    TriggL T1705,vl,laserOFF,z0,toolEtna\WObj:=wobjEtna;
    TriggL T1706,v50,laserON,z0,toolEtna\WObj:=wobjEtna;
    TriggL T1707,vl,laserOFF,z0,toolEtna\WObj:=wobjEtna;
    TriggL T1708,v50,laserON,z0,toolEtna\WObj:=wobjEtna;
    TriggL T1709,vl,laserOFF,z0,toolEtna\WObj:=wobjEtna;
    TriggL T1710,v50,laserON,z0,toolEtna\WObj:=wobjEtna;
    TriggL T1711,vl,laserOFF,z0,toolEtna\WObj:=wobjEtna;
    TriggL T1712,v50,laserON,z0,toolEtna\WObj:=wobjEtna;
    TriggL T1713,vl,laserOFF,z0,toolEtna\WObj:=wobjEtna;
    TriggL T1714,v50,laserON,z0,toolEtna\WObj:=wobjEtna;
    TriggL T1715,vl,laserOFF,z0,toolEtna\WObj:=wobjEtna;
    TriggL T1716,v50,laserON,z0,toolEtna\WObj:=wobjEtna;
    TriggL T1717,vl,laserOFF,z0,toolEtna\WObj:=wobjEtna;
    TriggL T1718,v50,laserON,z0,toolEtna\WObj:=wobjEtna;
    TriggL T1719,vl,laserOFF,z0,toolEtna\WObj:=wobjEtna;
    TriggL T1720,v50,laserON,z0,toolEtna\WObj:=wobjEtna;
    TriggL T1721,vl,laserOFF,z0,toolEtna\WObj:=wobjEtna;
    TriggL T1722,v50,laserON,z0,toolEtna\WObj:=wobjEtna;
    TriggL T1723,vl,laserOFF,z0,toolEtna\WObj:=wobjEtna;
    TriggL T1724,v50,laserON,z0,toolEtna\WObj:=wobjEtna;
    TriggL T1725,vl,laserOFF,z0,toolEtna\WObj:=wobjEtna;
    TriggL T1726,v50,laserON,z0,toolEtna\WObj:=wobjEtna;
    TriggL T1727,vl,laserOFF,z0,toolEtna\WObj:=wobjEtna;
    TriggL T1728,v50,laserON,z0,toolEtna\WObj:=wobjEtna;
    TriggL T1729,vl,laserOFF,z0,toolEtna\WObj:=wobjEtna;
    TriggL T1730,v50,laserON,z0,toolEtna\WObj:=wobjEtna;
    TriggL T1731,vl,laserOFF,z0,toolEtna\WObj:=wobjEtna;
    TriggL T1732,v50,laserON,z0,toolEtna\WObj:=wobjEtna;
    TriggL T1733,vl,laserOFF,z0,toolEtna\WObj:=wobjEtna;
    TriggL T1734,v50,laserON,z0,toolEtna\WObj:=wobjEtna;
    TriggL T1735,vl,laserOFF,z0,toolEtna\WObj:=wobjEtna;
    TriggL T1736,v50,laserON,z0,toolEtna\WObj:=wobjEtna;
    TriggL T1737,vl,laserOFF,z0,toolEtna\WObj:=wobjEtna;
    TriggL T1738,v50,laserON,z0,toolEtna\WObj:=wobjEtna;
    TriggL T1739,vl,laserOFF,z0,toolEtna\WObj:=wobjEtna;
    TriggL T1740,v50,laserON,z0,toolEtna\WObj:=wobjEtna;
    TriggL T1741,vl,laserOFF,z0,toolEtna\WObj:=wobjEtna;
    TriggL T1742,v50,laserON,z0,toolEtna\WObj:=wobjEtna;
    TriggL T1743,vl,laserOFF,z0,toolEtna\WObj:=wobjEtna;
    TriggL T1744,v50,laserON,z0,toolEtna\WObj:=wobjEtna;
    TriggL T1745,vl,laserOFF,z0,toolEtna\WObj:=wobjEtna;
    TriggL T1746,v50,laserON,z0,toolEtna\WObj:=wobjEtna;
    TriggL T1747,vl,laserOFF,z0,toolEtna\WObj:=wobjEtna;
    TriggL T1748,v50,laserON,z0,toolEtna\WObj:=wobjEtna;
    TriggL T1749,vl,laserOFF,z0,toolEtna\WObj:=wobjEtna;
    TriggL T1750,v50,laserON,z0,toolEtna\WObj:=wobjEtna;
    TriggL T1751,vl,laserOFF,z0,toolEtna\WObj:=wobjEtna;
    TriggL T1752,v50,laserON,z0,toolEtna\WObj:=wobjEtna;
    TriggL T1753,vl,laserOFF,z0,toolEtna\WObj:=wobjEtna;
    TriggL T1754,v50,laserON,z0,toolEtna\WObj:=wobjEtna;
    TriggL T1755,vl,laserOFF,z0,toolEtna\WObj:=wobjEtna;
    TriggL T1756,v50,laserON,z0,toolEtna\WObj:=wobjEtna;
    TriggL T1757,vl,laserOFF,z0,toolEtna\WObj:=wobjEtna;
    TriggL T1758,v50,laserON,z0,toolEtna\WObj:=wobjEtna;
    TriggL T1759,vl,laserOFF,z0,toolEtna\WObj:=wobjEtna;
    TriggL T1760,v50,laserON,z0,toolEtna\WObj:=wobjEtna;
    TriggL T1761,vl,laserOFF,z0,toolEtna\WObj:=wobjEtna;
    TriggL T1762,v50,laserON,z0,toolEtna\WObj:=wobjEtna;
    TriggL T1763,vl,laserOFF,z0,toolEtna\WObj:=wobjEtna;
    TriggL T1764,v50,laserON,z0,toolEtna\WObj:=wobjEtna;
    TriggL T1765,vl,laserOFF,z0,toolEtna\WObj:=wobjEtna;
    TriggL T1766,v50,laserON,z0,toolEtna\WObj:=wobjEtna;
    TriggL T1767,vl,laserOFF,z0,toolEtna\WObj:=wobjEtna;
    TriggL T1768,v50,laserON,z0,toolEtna\WObj:=wobjEtna;
    TriggL T1769,vl,laserOFF,z0,toolEtna\WObj:=wobjEtna;
    TriggL T1770,v50,laserON,z0,toolEtna\WObj:=wobjEtna;
    TriggL T1771,vl,laserOFF,z0,toolEtna\WObj:=wobjEtna;
    TriggL T1772,v50,laserON,z0,toolEtna\WObj:=wobjEtna;
    TriggL T1773,vl,laserOFF,z0,toolEtna\WObj:=wobjEtna;
    TriggL T1774,v50,laserON,z0,toolEtna\WObj:=wobjEtna;
    TriggL T1775,vl,laserOFF,z0,toolEtna\WObj:=wobjEtna;
    TriggL T1776,v50,laserON,z0,toolEtna\WObj:=wobjEtna;
    TriggL T1777,vl,laserOFF,z0,toolEtna\WObj:=wobjEtna;
    TriggL T1778,v50,laserON,z0,toolEtna\WObj:=wobjEtna;
    TriggL T1779,vl,laserOFF,z0,toolEtna\WObj:=wobjEtna;
    TriggL T1780,v50,laserON,z0,toolEtna\WObj:=wobjEtna;
    TriggL T1781,vl,laserOFF,z0,toolEtna\WObj:=wobjEtna;
    TriggL T1782,v50,laserON,z0,toolEtna\WObj:=wobjEtna;
    TriggL T1783,vl,laserOFF,z0,toolEtna\WObj:=wobjEtna;
    TriggL T1784,v50,laserON,z0,toolEtna\WObj:=wobjEtna;
    TriggL T1785,vl,laserOFF,z0,toolEtna\WObj:=wobjEtna;
    TriggL T1786,v50,laserON,z0,toolEtna\WObj:=wobjEtna;
    TriggL T1787,vl,laserOFF,z0,toolEtna\WObj:=wobjEtna;
    TriggL T1788,v50,laserON,z0,toolEtna\WObj:=wobjEtna;
    TriggL T1789,vl,laserOFF,z0,toolEtna\WObj:=wobjEtna;
    TriggL T1790,v50,laserON,z0,toolEtna\WObj:=wobjEtna;
    TriggL T1791,vl,laserOFF,z0,toolEtna\WObj:=wobjEtna;
    TriggL T1792,v50,laserON,z0,toolEtna\WObj:=wobjEtna;
    TriggL T1793,vl,laserOFF,z0,toolEtna\WObj:=wobjEtna;
    TriggL T1794,v50,laserON,z0,toolEtna\WObj:=wobjEtna;
    TriggL T1795,vl,laserOFF,z0,toolEtna\WObj:=wobjEtna;
    TriggL T1796,v50,laserON,z0,toolEtna\WObj:=wobjEtna;
    TriggL T1797,vl,laserOFF,z0,toolEtna\WObj:=wobjEtna;
    TriggL T1798,v50,laserON,z0,toolEtna\WObj:=wobjEtna;
    TriggL T1799,vl,laserOFF,z0,toolEtna\WObj:=wobjEtna;
    TriggL T1800,v50,laserON,z0,toolEtna\WObj:=wobjEtna;
    TriggL T1801,vl,laserOFF,z0,toolEtna\WObj:=wobjEtna;
    TriggL T1802,v50,laserON,z0,toolEtna\WObj:=wobjEtna;
    TriggL T1803,vl,laserOFF,z0,toolEtna\WObj:=wobjEtna;
    TriggL T1804,v50,laserON,z0,toolEtna\WObj:=wobjEtna;
    TriggL T1805,vl,laserOFF,z0,toolEtna\WObj:=wobjEtna;
    TriggL T1806,v50,laserON,z0,toolEtna\WObj:=wobjEtna;
    TriggL T1807,vl,laserOFF,z0,toolEtna\WObj:=wobjEtna;
    TriggL T1808,v50,laserON,z0,toolEtna\WObj:=wobjEtna;
    TriggL T1809,vl,laserOFF,z0,toolEtna\WObj:=wobjEtna;
    TriggL T1810,v50,laserON,z0,toolEtna\WObj:=wobjEtna;
    TriggL T1811,vl,laserOFF,z0,toolEtna\WObj:=wobjEtna;
    TriggL T1812,v50,laserON,z0,toolEtna\WObj:=wobjEtna;
    TriggL T1813,vl,laserOFF,z0,toolEtna\WObj:=wobjEtna;
    TriggL T1814,v50,laserON,z0,toolEtna\WObj:=wobjEtna;
    TriggL T1815,vl,laserOFF,z0,toolEtna\WObj:=wobjEtna;
    TriggL T1816,v50,laserON,z0,toolEtna\WObj:=wobjEtna;
    TriggL T1817,vl,laserOFF,z0,toolEtna\WObj:=wobjEtna;
    TriggL T1818,v50,laserON,z0,toolEtna\WObj:=wobjEtna;
    TriggL T1819,vl,laserOFF,z0,toolEtna\WObj:=wobjEtna;
    TriggL T1820,v50,laserON,z0,toolEtna\WObj:=wobjEtna;
    TriggL T1821,vl,laserOFF,z0,toolEtna\WObj:=wobjEtna;
    TriggL T1822,v50,laserON,z0,toolEtna\WObj:=wobjEtna;
    TriggL T1823,vl,laserOFF,z0,toolEtna\WObj:=wobjEtna;
    TriggL T1824,v50,laserON,z0,toolEtna\WObj:=wobjEtna;
    TriggL T1825,vl,laserOFF,z0,toolEtna\WObj:=wobjEtna;
    TriggL T1826,v50,laserON,z0,toolEtna\WObj:=wobjEtna;
    TriggL T1827,vl,laserOFF,z0,toolEtna\WObj:=wobjEtna;
    TriggL T1828,v50,laserON,z0,toolEtna\WObj:=wobjEtna;
    TriggL T1829,vl,laserOFF,z0,toolEtna\WObj:=wobjEtna;
    TriggL T1830,v50,laserON,z0,toolEtna\WObj:=wobjEtna;
    TriggL T1831,vl,laserOFF,z0,toolEtna\WObj:=wobjEtna;
    TriggL T1832,v50,laserON,z0,toolEtna\WObj:=wobjEtna;
    TriggL T1833,vl,laserOFF,z0,toolEtna\WObj:=wobjEtna;
    TriggL T1834,v50,laserON,z0,toolEtna\WObj:=wobjEtna;
    TriggL T1835,vl,laserOFF,z0,toolEtna\WObj:=wobjEtna;
    TriggL T1836,v50,laserON,z0,toolEtna\WObj:=wobjEtna;
    TriggL T1837,vl,laserOFF,z0,toolEtna\WObj:=wobjEtna;
    TriggL T1838,v50,laserON,z0,toolEtna\WObj:=wobjEtna;
    TriggL T1839,vl,laserOFF,z0,toolEtna\WObj:=wobjEtna;
    TriggL T1840,v50,laserON,z0,toolEtna\WObj:=wobjEtna;
    TriggL T1841,vl,laserOFF,z0,toolEtna\WObj:=wobjEtna;
    TriggL T1842,v50,laserON,z0,toolEtna\WObj:=wobjEtna;
    TriggL T1843,vl,laserOFF,z0,toolEtna\WObj:=wobjEtna;
    TriggL T1844,v50,laserON,z0,toolEtna\WObj:=wobjEtna;
    TriggL T1845,vl,laserOFF,z0,toolEtna\WObj:=wobjEtna;
    TriggL T1846,v50,laserON,z0,toolEtna\WObj:=wobjEtna;
    TriggL T1847,vl,laserOFF,z0,toolEtna\WObj:=wobjEtna;
    TriggL T1848,v50,laserON,z0,toolEtna\WObj:=wobjEtna;
    TriggL T1849,vl,laserOFF,z0,toolEtna\WObj:=wobjEtna;
    TriggL T1850,v50,laserON,z0,toolEtna\WObj:=wobjEtna;
    TriggL T1851,vl,laserOFF,z0,toolEtna\WObj:=wobjEtna;
    TriggL T1852,v50,laserON,z0,toolEtna\WObj:=wobjEtna;
    TriggL T1853,vl,laserOFF,z0,toolEtna\WObj:=wobjEtna;
    TriggL T1854,v50,laserON,z0,toolEtna\WObj:=wobjEtna;
    TriggL T1855,vl,laserOFF,z0,toolEtna\WObj:=wobjEtna;
    TriggL T1856,v50,laserON,z0,toolEtna\WObj:=wobjEtna;
    TriggL T1857,vl,laserOFF,z0,toolEtna\WObj:=wobjEtna;
    TriggL T1858,v50,laserON,z0,toolEtna\WObj:=wobjEtna;
    TriggL T1859,vl,laserOFF,z0,toolEtna\WObj:=wobjEtna;
    TriggL T1860,v50,laserON,z0,toolEtna\WObj:=wobjEtna;
    TriggL T1861,vl,laserOFF,z0,toolEtna\WObj:=wobjEtna;
    TriggL T1862,v50,laserON,z0,toolEtna\WObj:=wobjEtna;
    TriggL T1863,vl,laserOFF,z0,toolEtna\WObj:=wobjEtna;
    TriggL T1864,v50,laserON,z0,toolEtna\WObj:=wobjEtna;
    TriggL T1865,vl,laserOFF,z0,toolEtna\WObj:=wobjEtna;
    TriggL T1866,v50,laserON,z0,toolEtna\WObj:=wobjEtna;
    TriggL T1867,vl,laserOFF,z0,toolEtna\WObj:=wobjEtna;
    TriggL T1868,v50,laserON,z0,toolEtna\WObj:=wobjEtna;
    TriggL T1869,vl,laserOFF,z0,toolEtna\WObj:=wobjEtna;
    TriggL T1870,v50,laserON,z0,toolEtna\WObj:=wobjEtna;
    TriggL T1871,vl,laserOFF,z0,toolEtna\WObj:=wobjEtna;
    TriggL T1872,v50,laserON,z0,toolEtna\WObj:=wobjEtna;
    TriggL T1873,vl,laserOFF,z0,toolEtna\WObj:=wobjEtna;
    TriggL T1874,v50,laserON,z0,toolEtna\WObj:=wobjEtna;
    TriggL T1875,vl,laserOFF,z0,toolEtna\WObj:=wobjEtna;
    TriggL T1876,v50,laserON,z0,toolEtna\WObj:=wobjEtna;
    TriggL T1877,vl,laserOFF,z0,toolEtna\WObj:=wobjEtna;
    TriggL T1878,v50,laserON,z0,toolEtna\WObj:=wobjEtna;
    TriggL T1879,vl,laserOFF,z0,toolEtna\WObj:=wobjEtna;
    TriggL T1880,v50,laserON,z0,toolEtna\WObj:=wobjEtna;
    TriggL T1881,vl,laserOFF,z0,toolEtna\WObj:=wobjEtna;
    TriggL T1882,v50,laserON,z0,toolEtna\WObj:=wobjEtna;
    TriggL T1883,vl,laserOFF,z0,toolEtna\WObj:=wobjEtna;
    TriggL T1884,v50,laserON,z0,toolEtna\WObj:=wobjEtna;
    TriggL T1885,vl,laserOFF,z0,toolEtna\WObj:=wobjEtna;
    TriggL T1886,v50,laserON,z0,toolEtna\WObj:=wobjEtna;
    TriggL T1887,vl,laserOFF,z0,toolEtna\WObj:=wobjEtna;
    TriggL T1888,v50,laserON,z0,toolEtna\WObj:=wobjEtna;
    TriggL T1889,vl,laserOFF,z0,toolEtna\WObj:=wobjEtna;
    TriggL T1890,v50,laserON,z0,toolEtna\WObj:=wobjEtna;
    TriggL T1891,vl,laserOFF,z0,toolEtna\WObj:=wobjEtna;
    TriggL T1892,v50,laserON,z0,toolEtna\WObj:=wobjEtna;
    TriggL T1893,vl,laserOFF,z0,toolEtna\WObj:=wobjEtna;
    TriggL T1894,v50,laserON,z0,toolEtna\WObj:=wobjEtna;
    TriggL T1895,vl,laserOFF,z0,toolEtna\WObj:=wobjEtna;
    TriggL T1896,v50,laserON,z0,toolEtna\WObj:=wobjEtna;
    TriggL T1897,vl,laserOFF,z0,toolEtna\WObj:=wobjEtna;
    TriggL T1898,v50,laserON,z0,toolEtna\WObj:=wobjEtna;
    TriggL T1899,vl,laserOFF,z0,toolEtna\WObj:=wobjEtna;
    TriggL T1900,v50,laserON,z0,toolEtna\WObj:=wobjEtna;
    TriggL T1901,vl,laserOFF,z0,toolEtna\WObj:=wobjEtna;
    TriggL T1902,v50,laserON,z0,toolEtna\WObj:=wobjEtna;
    TriggL T1903,vl,laserOFF,z0,toolEtna\WObj:=wobjEtna;
    TriggL T1904,v50,laserON,z0,toolEtna\WObj:=wobjEtna;
    TriggL T1905,vl,laserOFF,z0,toolEtna\WObj:=wobjEtna;
    TriggL T1906,v50,laserON,z0,toolEtna\WObj:=wobjEtna;
    TriggL T1907,vl,laserOFF,z0,toolEtna\WObj:=wobjEtna;
    TriggL T1908,v50,laserON,z0,toolEtna\WObj:=wobjEtna;
    TriggL T1909,vl,laserOFF,z0,toolEtna\WObj:=wobjEtna;
    TriggL T1910,v50,laserON,z0,toolEtna\WObj:=wobjEtna;
    TriggL T1911,vl,laserOFF,z0,toolEtna\WObj:=wobjEtna;
    TriggL T1912,v50,laserON,z0,toolEtna\WObj:=wobjEtna;
    TriggL T1913,vl,laserOFF,z0,toolEtna\WObj:=wobjEtna;
    TriggL T1914,v50,laserON,z0,toolEtna\WObj:=wobjEtna;
    TriggL T1915,vl,laserOFF,z0,toolEtna\WObj:=wobjEtna;
    TriggL T1916,v50,laserON,z0,toolEtna\WObj:=wobjEtna;
    TriggL T1917,vl,laserOFF,z0,toolEtna\WObj:=wobjEtna;
    TriggL T1918,v50,laserON,z0,toolEtna\WObj:=wobjEtna;
    TriggL T1919,vl,laserOFF,z0,toolEtna\WObj:=wobjEtna;
    TriggL T1920,v50,laserON,z0,toolEtna\WObj:=wobjEtna;
    TriggL T1921,vl,laserOFF,z0,toolEtna\WObj:=wobjEtna;
    TriggL T1922,v50,laserON,z0,toolEtna\WObj:=wobjEtna;
    TriggL T1923,vl,laserOFF,z0,toolEtna\WObj:=wobjEtna;
    TriggL T1924,v50,laserON,z0,toolEtna\WObj:=wobjEtna;
    TriggL T1925,vl,laserOFF,z0,toolEtna\WObj:=wobjEtna;
    TriggL T1926,v50,laserON,z0,toolEtna\WObj:=wobjEtna;
    TriggL T1927,vl,laserOFF,z0,toolEtna\WObj:=wobjEtna;
    TriggL T1928,v50,laserON,z0,toolEtna\WObj:=wobjEtna;
    TriggL T1929,vl,laserOFF,z0,toolEtna\WObj:=wobjEtna;
    TriggL T1930,v50,laserON,z0,toolEtna\WObj:=wobjEtna;
    TriggL T1931,vl,laserOFF,z0,toolEtna\WObj:=wobjEtna;
    TriggL T1932,v50,laserON,z0,toolEtna\WObj:=wobjEtna;
    TriggL T1933,vl,laserOFF,z0,toolEtna\WObj:=wobjEtna;
    TriggL T1934,v50,laserON,z0,toolEtna\WObj:=wobjEtna;
    TriggL T1935,vl,laserOFF,z0,toolEtna\WObj:=wobjEtna;
    TriggL T1936,v50,laserON,z0,toolEtna\WObj:=wobjEtna;
    TriggL T1937,vl,laserOFF,z0,toolEtna\WObj:=wobjEtna;
    TriggL T1938,v50,laserON,z0,toolEtna\WObj:=wobjEtna;
    TriggL T1939,vl,laserOFF,z0,toolEtna\WObj:=wobjEtna;
    TriggL T1940,v50,laserON,z0,toolEtna\WObj:=wobjEtna;
    TriggL T1941,vl,laserOFF,z0,toolEtna\WObj:=wobjEtna;
    TriggL T1942,v50,laserON,z0,toolEtna\WObj:=wobjEtna;
    TriggL T1943,vl,laserOFF,z0,toolEtna\WObj:=wobjEtna;
    TriggL T1944,v50,laserON,z0,toolEtna\WObj:=wobjEtna;
    TriggL T1945,vl,laserOFF,z0,toolEtna\WObj:=wobjEtna;
    TriggL T1946,v50,laserON,z0,toolEtna\WObj:=wobjEtna;
    TriggL T1947,vl,laserOFF,z0,toolEtna\WObj:=wobjEtna;
    TriggL T1948,v50,laserON,z0,toolEtna\WObj:=wobjEtna;
    TriggL T1949,vl,laserOFF,z0,toolEtna\WObj:=wobjEtna;
    TriggL T1950,v50,laserON,z0,toolEtna\WObj:=wobjEtna;
    TriggL T1951,vl,laserOFF,z0,toolEtna\WObj:=wobjEtna;
    TriggL T1952,v50,laserON,z0,toolEtna\WObj:=wobjEtna;
    TriggL T1953,vl,laserOFF,z0,toolEtna\WObj:=wobjEtna;
    TriggL T1954,v50,laserON,z0,toolEtna\WObj:=wobjEtna;
    TriggL T1955,vl,laserOFF,z0,toolEtna\WObj:=wobjEtna;
    TriggL T1956,v50,laserON,z0,toolEtna\WObj:=wobjEtna;
    TriggL T1957,vl,laserOFF,z0,toolEtna\WObj:=wobjEtna;
    TriggL T1958,v50,laserON,z0,toolEtna\WObj:=wobjEtna;
    TriggL T1959,vl,laserOFF,z0,toolEtna\WObj:=wobjEtna;
    TriggL T1960,v50,laserON,z0,toolEtna\WObj:=wobjEtna;
    TriggL T1961,vl,laserOFF,z0,toolEtna\WObj:=wobjEtna;
    TriggL T1962,v50,laserON,z0,toolEtna\WObj:=wobjEtna;
    TriggL T1963,vl,laserOFF,z0,toolEtna\WObj:=wobjEtna;
    TriggL T1964,v50,laserON,z0,toolEtna\WObj:=wobjEtna;
    TriggL T1965,vl,laserOFF,z0,toolEtna\WObj:=wobjEtna;
    TriggL T1966,v50,laserON,z0,toolEtna\WObj:=wobjEtna;
    TriggL T1967,vl,laserOFF,z0,toolEtna\WObj:=wobjEtna;
    TriggL T1968,v50,laserON,z0,toolEtna\WObj:=wobjEtna;
    TriggL T1969,vl,laserOFF,z0,toolEtna\WObj:=wobjEtna;
    TriggL T1970,v50,laserON,z0,toolEtna\WObj:=wobjEtna;
    TriggL T1971,vl,laserOFF,z0,toolEtna\WObj:=wobjEtna;
    TriggL T1972,v50,laserON,z0,toolEtna\WObj:=wobjEtna;
    TriggL T1973,vl,laserOFF,z0,toolEtna\WObj:=wobjEtna;
    TriggL T1974,v50,laserON,z0,toolEtna\WObj:=wobjEtna;
    TriggL T1975,vl,laserOFF,z0,toolEtna\WObj:=wobjEtna;
    TriggL T1976,v50,laserON,z0,toolEtna\WObj:=wobjEtna;
    TriggL T1977,vl,laserOFF,z0,toolEtna\WObj:=wobjEtna;
    TriggL T1978,v50,laserON,z0,toolEtna\WObj:=wobjEtna;
    TriggL T1979,vl,laserOFF,z0,toolEtna\WObj:=wobjEtna;
    TriggL T1980,v50,laserON,z0,toolEtna\WObj:=wobjEtna;
    TriggL T1981,vl,laserOFF,z0,toolEtna\WObj:=wobjEtna;
    TriggL T1982,v50,laserON,z0,toolEtna\WObj:=wobjEtna;
    TriggL T1983,vl,laserOFF,z0,toolEtna\WObj:=wobjEtna;
    TriggL T1984,v50,laserON,z0,toolEtna\WObj:=wobjEtna;
    TriggL T1985,vl,laserOFF,z0,toolEtna\WObj:=wobjEtna;
    TriggL T1986,v50,laserON,z0,toolEtna\WObj:=wobjEtna;
    TriggL T1987,vl,laserOFF,z0,toolEtna\WObj:=wobjEtna;
    TriggL T1988,v50,laserON,z0,toolEtna\WObj:=wobjEtna;
    TriggL T1989,vl,laserOFF,z0,toolEtna\WObj:=wobjEtna;
    TriggL T1990,v50,laserON,z0,toolEtna\WObj:=wobjEtna;
    TriggL T1991,vl,laserOFF,z0,toolEtna\WObj:=wobjEtna;
    TriggL T1992,v50,laserON,z0,toolEtna\WObj:=wobjEtna;
    TriggL T1993,vl,laserOFF,z0,toolEtna\WObj:=wobjEtna;
    TriggL T1994,v50,laserON,z0,toolEtna\WObj:=wobjEtna;
    TriggL T1995,vl,laserOFF,z0,toolEtna\WObj:=wobjEtna;
    TriggL T1996,v50,laserON,z0,toolEtna\WObj:=wobjEtna;
    TriggL T1997,vl,laserOFF,z0,toolEtna\WObj:=wobjEtna;
    TriggL T1998,v50,laserON,z0,toolEtna\WObj:=wobjEtna;
    TriggL T1999,vl,laserOFF,z0,toolEtna\WObj:=wobjEtna;
    TriggL T2000,v50,laserON,z0,toolEtna\WObj:=wobjEtna;
    TriggL T2001,vl,laserOFF,z0,toolEtna\WObj:=wobjEtna;
    TriggL T2002,v50,laserON,z0,toolEtna\WObj:=wobjEtna;
    TriggL T2003,vl,laserOFF,z0,toolEtna\WObj:=wobjEtna;
    TriggL T2004,v50,laserON,z0,toolEtna\WObj:=wobjEtna;
    TriggL T2005,vl,laserOFF,z0,toolEtna\WObj:=wobjEtna;
    TriggL T2006,v50,laserON,z0,toolEtna\WObj:=wobjEtna;
    TriggL T2007,vl,laserOFF,z0,toolEtna\WObj:=wobjEtna;
    TriggL T2008,v50,laserON,z0,toolEtna\WObj:=wobjEtna;
    TriggL T2009,vl,laserOFF,z0,toolEtna\WObj:=wobjEtna;
    TriggL T2010,v50,laserON,z0,toolEtna\WObj:=wobjEtna;
    TriggL T2011,vl,laserOFF,z0,toolEtna\WObj:=wobjEtna;
    TriggL T2012,v50,laserON,z0,toolEtna\WObj:=wobjEtna;
    TriggL T2013,vl,laserOFF,z0,toolEtna\WObj:=wobjEtna;
    TriggL T2014,v50,laserON,z0,toolEtna\WObj:=wobjEtna;
    TriggL T2015,vl,laserOFF,z0,toolEtna\WObj:=wobjEtna;
    TriggL T2016,v50,laserON,z0,toolEtna\WObj:=wobjEtna;
    TriggL T2017,vl,laserOFF,z0,toolEtna\WObj:=wobjEtna;
    TriggL T2018,v50,laserON,z0,toolEtna\WObj:=wobjEtna;
    TriggL T2019,vl,laserOFF,z0,toolEtna\WObj:=wobjEtna;
    TriggL T2020,v50,laserON,z0,toolEtna\WObj:=wobjEtna;
    TriggL T2021,vl,laserOFF,z0,toolEtna\WObj:=wobjEtna;
    TriggL T2022,v50,laserON,z0,toolEtna\WObj:=wobjEtna;
    TriggL T2023,vl,laserOFF,z0,toolEtna\WObj:=wobjEtna;
    TriggL T2024,v50,laserON,z0,toolEtna\WObj:=wobjEtna;
    TriggL T2025,vl,laserOFF,z0,toolEtna\WObj:=wobjEtna;
    TriggL T2026,v50,laserON,z0,toolEtna\WObj:=wobjEtna;
    TriggL T2027,vl,laserOFF,z0,toolEtna\WObj:=wobjEtna;
    TriggL T2028,v50,laserON,z0,toolEtna\WObj:=wobjEtna;
    TriggL T2029,vl,laserOFF,z0,toolEtna\WObj:=wobjEtna;
    TriggL T2030,v50,laserON,z0,toolEtna\WObj:=wobjEtna;
    TriggL T2031,vl,laserOFF,z0,toolEtna\WObj:=wobjEtna;
    TriggL T2032,v50,laserON,z0,toolEtna\WObj:=wobjEtna;
    TriggL T2033,vl,laserOFF,z0,toolEtna\WObj:=wobjEtna;
    TriggL T2034,v50,laserON,z0,toolEtna\WObj:=wobjEtna;
    TriggL T2035,vl,laserOFF,z0,toolEtna\WObj:=wobjEtna;
    TriggL T2036,v50,laserON,z0,toolEtna\WObj:=wobjEtna;
    TriggL T2037,vl,laserOFF,z0,toolEtna\WObj:=wobjEtna;
    TriggL T2038,v50,laserON,z0,toolEtna\WObj:=wobjEtna;
    TriggL T2039,vl,laserOFF,z0,toolEtna\WObj:=wobjEtna;
    TriggL T2040,v50,laserON,z0,toolEtna\WObj:=wobjEtna;
    TriggL T2041,vl,laserOFF,z0,toolEtna\WObj:=wobjEtna;
    TriggL T2042,v50,laserON,z0,toolEtna\WObj:=wobjEtna;
    TriggL T2043,vl,laserOFF,z0,toolEtna\WObj:=wobjEtna;
    TriggL T2044,v50,laserON,z0,toolEtna\WObj:=wobjEtna;
    TriggL T2045,vl,laserOFF,z0,toolEtna\WObj:=wobjEtna;
    TriggL T2046,v50,laserON,z0,toolEtna\WObj:=wobjEtna;
    TriggL T2047,vl,laserOFF,z0,toolEtna\WObj:=wobjEtna;
    TriggL T2048,v50,laserON,z0,toolEtna\WObj:=wobjEtna;
    TriggL T2049,vl,laserOFF,z0,toolEtna\WObj:=wobjEtna;
    TriggL T2050,v50,laserON,z0,toolEtna\WObj:=wobjEtna;
    TriggL T2051,vl,laserOFF,z0,toolEtna\WObj:=wobjEtna;
    TriggL T2052,v50,laserON,z0,toolEtna\WObj:=wobjEtna;
    TriggL T2053,vl,laserOFF,z0,toolEtna\WObj:=wobjEtna;
    TriggL T2054,v50,laserON,z0,toolEtna\WObj:=wobjEtna;
    TriggL T2055,vl,laserOFF,z0,toolEtna\WObj:=wobjEtna;
    TriggL T2056,v50,laserON,z0,toolEtna\WObj:=wobjEtna;
    TriggL T2057,vl,laserOFF,z0,toolEtna\WObj:=wobjEtna;
    TriggL T2058,v50,laserON,z0,toolEtna\WObj:=wobjEtna;
    TriggL T2059,vl,laserOFF,z0,toolEtna\WObj:=wobjEtna;
    TriggL T2060,v50,laserON,z0,toolEtna\WObj:=wobjEtna;
    TriggL T2061,vl,laserOFF,z0,toolEtna\WObj:=wobjEtna;
    TriggL T2062,v50,laserON,z0,toolEtna\WObj:=wobjEtna;
    TriggL T2063,vl,laserOFF,z0,toolEtna\WObj:=wobjEtna;
    TriggL T2064,v50,laserON,z0,toolEtna\WObj:=wobjEtna;
    TriggL T2065,vl,laserOFF,z0,toolEtna\WObj:=wobjEtna;
    TriggL T2066,v50,laserON,z0,toolEtna\WObj:=wobjEtna;
    TriggL T2067,vl,laserOFF,z0,toolEtna\WObj:=wobjEtna;
    TriggL T2068,v50,laserON,z0,toolEtna\WObj:=wobjEtna;
    TriggL T2069,vl,laserOFF,z0,toolEtna\WObj:=wobjEtna;
    TriggL T2070,v50,laserON,z0,toolEtna\WObj:=wobjEtna;
    TriggL T2071,vl,laserOFF,z0,toolEtna\WObj:=wobjEtna;
    TriggL T2072,v50,laserON,z0,toolEtna\WObj:=wobjEtna;
    TriggL T2073,vl,laserOFF,z0,toolEtna\WObj:=wobjEtna;
    TriggL T2074,v50,laserON,z0,toolEtna\WObj:=wobjEtna;
    TriggL T2075,vl,laserOFF,z0,toolEtna\WObj:=wobjEtna;
    TriggL T2076,v50,laserON,z0,toolEtna\WObj:=wobjEtna;
    TriggL T2077,vl,laserOFF,z0,toolEtna\WObj:=wobjEtna;
    TriggL T2078,v50,laserON,z0,toolEtna\WObj:=wobjEtna;
    TriggL T2079,vl,laserOFF,z0,toolEtna\WObj:=wobjEtna;
    TriggL T2080,v50,laserON,z0,toolEtna\WObj:=wobjEtna;
    TriggL T2081,vl,laserOFF,z0,toolEtna\WObj:=wobjEtna;
    TriggL T2082,v50,laserON,z0,toolEtna\WObj:=wobjEtna;
    TriggL T2083,vl,laserOFF,z0,toolEtna\WObj:=wobjEtna;
    TriggL T2084,v50,laserON,z0,toolEtna\WObj:=wobjEtna;
    TriggL T2085,vl,laserOFF,z0,toolEtna\WObj:=wobjEtna;
    TriggL T2086,v50,laserON,z0,toolEtna\WObj:=wobjEtna;
    TriggL T2087,vl,laserOFF,z0,toolEtna\WObj:=wobjEtna;
    TriggL T2088,v50,laserON,z0,toolEtna\WObj:=wobjEtna;
    TriggL T2089,vl,laserOFF,z0,toolEtna\WObj:=wobjEtna;
    TriggL T2090,v50,laserON,z0,toolEtna\WObj:=wobjEtna;
    TriggL T2091,vl,laserOFF,z0,toolEtna\WObj:=wobjEtna;
    TriggL T2092,v50,laserON,z0,toolEtna\WObj:=wobjEtna;
    TriggL T2093,vl,laserOFF,z0,toolEtna\WObj:=wobjEtna;
    TriggL T2094,v50,laserON,z0,toolEtna\WObj:=wobjEtna;
    TriggL T2095,vl,laserOFF,z0,toolEtna\WObj:=wobjEtna;
    TriggL T2096,v50,laserON,z0,toolEtna\WObj:=wobjEtna;
    TriggL T2097,vl,laserOFF,z0,toolEtna\WObj:=wobjEtna;
    TriggL T2098,v50,laserON,z0,toolEtna\WObj:=wobjEtna;
    TriggL T2099,vl,laserOFF,z0,toolEtna\WObj:=wobjEtna;
    TriggL T2100,v50,laserON,z0,toolEtna\WObj:=wobjEtna;
    TriggL T2101,vl,laserOFF,z0,toolEtna\WObj:=wobjEtna;
    TriggL T2102,v50,laserON,z0,toolEtna\WObj:=wobjEtna;
    TriggL T2103,vl,laserOFF,z0,toolEtna\WObj:=wobjEtna;
    TriggL T2104,v50,laserON,z0,toolEtna\WObj:=wobjEtna;
    TriggL T2105,vl,laserOFF,z0,toolEtna\WObj:=wobjEtna;
    TriggL T2106,v50,laserON,z0,toolEtna\WObj:=wobjEtna;
    TriggL T2107,vl,laserOFF,z0,toolEtna\WObj:=wobjEtna;
    TriggL T2108,v50,laserON,z0,toolEtna\WObj:=wobjEtna;
    TriggL T2109,vl,laserOFF,z0,toolEtna\WObj:=wobjEtna;
    TriggL T2110,v50,laserON,z0,toolEtna\WObj:=wobjEtna;
    TriggL T2111,vl,laserOFF,z0,toolEtna\WObj:=wobjEtna;
    TriggL T2112,v50,laserON,z0,toolEtna\WObj:=wobjEtna;
    TriggL T2113,vl,laserOFF,z0,toolEtna\WObj:=wobjEtna;
    TriggL T2114,v50,laserON,z0,toolEtna\WObj:=wobjEtna;
    TriggL T2115,vl,laserOFF,z0,toolEtna\WObj:=wobjEtna;
    TriggL T2116,v50,laserON,z0,toolEtna\WObj:=wobjEtna;
    TriggL T2117,vl,laserOFF,z0,toolEtna\WObj:=wobjEtna;
    TriggL T2118,v50,laserON,z0,toolEtna\WObj:=wobjEtna;
    TriggL T2119,vl,laserOFF,z0,toolEtna\WObj:=wobjEtna;
    TriggL T2120,v50,laserON,z0,toolEtna\WObj:=wobjEtna;
    TriggL T2121,vl,laserOFF,z0,toolEtna\WObj:=wobjEtna;
    TriggL T2122,v50,laserON,z0,toolEtna\WObj:=wobjEtna;
    TriggL T2123,vl,laserOFF,z0,toolEtna\WObj:=wobjEtna;
    TriggL T2124,v50,laserON,z0,toolEtna\WObj:=wobjEtna;
    TriggL T2125,vl,laserOFF,z0,toolEtna\WObj:=wobjEtna;
    TriggL T2126,v50,laserON,z0,toolEtna\WObj:=wobjEtna;
    TriggL T2127,vl,laserOFF,z0,toolEtna\WObj:=wobjEtna;
    TriggL T2128,v50,laserON,z0,toolEtna\WObj:=wobjEtna;
    TriggL T2129,vl,laserOFF,z0,toolEtna\WObj:=wobjEtna;
    TriggL T2130,v50,laserON,z0,toolEtna\WObj:=wobjEtna;
    TriggL T2131,vl,laserOFF,z0,toolEtna\WObj:=wobjEtna;
    TriggL T2132,v50,laserON,z0,toolEtna\WObj:=wobjEtna;
    TriggL T2133,vl,laserOFF,z0,toolEtna\WObj:=wobjEtna;
    TriggL T2134,v50,laserON,z0,toolEtna\WObj:=wobjEtna;
    TriggL T2135,vl,laserOFF,z0,toolEtna\WObj:=wobjEtna;
    TriggL T2136,v50,laserON,z0,toolEtna\WObj:=wobjEtna;
    TriggL T2137,vl,laserOFF,z0,toolEtna\WObj:=wobjEtna;
    TriggL T2138,v50,laserON,z0,toolEtna\WObj:=wobjEtna;
    TriggL T2139,vl,laserOFF,z0,toolEtna\WObj:=wobjEtna;
    TriggL T2140,v50,laserON,z0,toolEtna\WObj:=wobjEtna;
    TriggL T2141,vl,laserOFF,z0,toolEtna\WObj:=wobjEtna;
    TriggL T2142,v50,laserON,z0,toolEtna\WObj:=wobjEtna;
    TriggL T2143,vl,laserOFF,z0,toolEtna\WObj:=wobjEtna;
    TriggL T2144,v50,laserON,z0,toolEtna\WObj:=wobjEtna;
    TriggL T2145,vl,laserOFF,z0,toolEtna\WObj:=wobjEtna;
    TriggL T2146,v50,laserON,z0,toolEtna\WObj:=wobjEtna;
    TriggL T2147,vl,laserOFF,z0,toolEtna\WObj:=wobjEtna;
    TriggL T2148,v50,laserON,z0,toolEtna\WObj:=wobjEtna;
    TriggL T2149,vl,laserOFF,z0,toolEtna\WObj:=wobjEtna;
    TriggL T2150,v50,laserON,z0,toolEtna\WObj:=wobjEtna;
    TriggL T2151,vl,laserOFF,z0,toolEtna\WObj:=wobjEtna;
    TriggL T2152,v50,laserON,z0,toolEtna\WObj:=wobjEtna;
    TriggL T2153,vl,laserOFF,z0,toolEtna\WObj:=wobjEtna;
    TriggL T2154,v50,laserON,z0,toolEtna\WObj:=wobjEtna;
    TriggL T2155,vl,laserOFF,z0,toolEtna\WObj:=wobjEtna;
    TriggL T2156,v50,laserON,z0,toolEtna\WObj:=wobjEtna;
    TriggL T2157,vl,laserOFF,z0,toolEtna\WObj:=wobjEtna;
    TriggL T2158,v50,laserON,z0,toolEtna\WObj:=wobjEtna;
    TriggL T2159,vl,laserOFF,z0,toolEtna\WObj:=wobjEtna;
    TriggL T2160,v50,laserON,z0,toolEtna\WObj:=wobjEtna;
    TriggL T2161,vl,laserOFF,z0,toolEtna\WObj:=wobjEtna;
    TriggL T2162,v50,laserON,z0,toolEtna\WObj:=wobjEtna;
    TriggL T2163,vl,laserOFF,z0,toolEtna\WObj:=wobjEtna;
    TriggL T2164,v50,laserON,z0,toolEtna\WObj:=wobjEtna;
    TriggL T2165,vl,laserOFF,z0,toolEtna\WObj:=wobjEtna;
    TriggL T2166,v50,laserON,z0,toolEtna\WObj:=wobjEtna;
    TriggL T2167,vl,laserOFF,z0,toolEtna\WObj:=wobjEtna;
    TriggL T2168,v50,laserON,z0,toolEtna\WObj:=wobjEtna;
    TriggL T2169,vl,laserOFF,z0,toolEtna\WObj:=wobjEtna;
    TriggL T2170,v50,laserON,z0,toolEtna\WObj:=wobjEtna;
    TriggL T2171,vl,laserOFF,z0,toolEtna\WObj:=wobjEtna;
    TriggL T2172,v50,laserON,z0,toolEtna\WObj:=wobjEtna;
    TriggL T2173,vl,laserOFF,z0,toolEtna\WObj:=wobjEtna;
    TriggL T2174,v50,laserON,z0,toolEtna\WObj:=wobjEtna;
    TriggL T2175,vl,laserOFF,z0,toolEtna\WObj:=wobjEtna;
    TriggL T2176,v50,laserON,z0,toolEtna\WObj:=wobjEtna;
    TriggL T2177,vl,laserOFF,z0,toolEtna\WObj:=wobjEtna;
    TriggL T2178,v50,laserON,z0,toolEtna\WObj:=wobjEtna;
    TriggL T2179,vl,laserOFF,z0,toolEtna\WObj:=wobjEtna;
    TriggL T2180,v50,laserON,z0,toolEtna\WObj:=wobjEtna;
    TriggL T2181,vl,laserOFF,z0,toolEtna\WObj:=wobjEtna;
    TriggL T2182,v50,laserON,z0,toolEtna\WObj:=wobjEtna;
    TriggL T2183,vl,laserOFF,z0,toolEtna\WObj:=wobjEtna;
    TriggL T2184,v50,laserON,z0,toolEtna\WObj:=wobjEtna;
    TriggL T2185,vl,laserOFF,z0,toolEtna\WObj:=wobjEtna;
    TriggL T2186,v50,laserON,z0,toolEtna\WObj:=wobjEtna;
    TriggL T2187,vl,laserOFF,z0,toolEtna\WObj:=wobjEtna;
    TriggL T2188,v50,laserON,z0,toolEtna\WObj:=wobjEtna;
    TriggL T2189,vl,laserOFF,z0,toolEtna\WObj:=wobjEtna;
    TriggL T2190,v50,laserON,z0,toolEtna\WObj:=wobjEtna;
    TriggL T2191,vl,laserOFF,z0,toolEtna\WObj:=wobjEtna;
    TriggL T2192,v50,laserON,z0,toolEtna\WObj:=wobjEtna;
    TriggL T2193,vl,laserOFF,z0,toolEtna\WObj:=wobjEtna;
    TriggL T2194,v50,laserON,z0,toolEtna\WObj:=wobjEtna;
    TriggL T2195,vl,laserOFF,z0,toolEtna\WObj:=wobjEtna;
    TriggL T2196,v50,laserON,z0,toolEtna\WObj:=wobjEtna;
    TriggL T2197,vl,laserOFF,z0,toolEtna\WObj:=wobjEtna;
    TriggL T2198,v50,laserON,z0,toolEtna\WObj:=wobjEtna;
    TriggL T2199,vl,laserOFF,z0,toolEtna\WObj:=wobjEtna;
    TriggL T2200,v50,laserON,z0,toolEtna\WObj:=wobjEtna;
    TriggL T2201,vl,laserOFF,z0,toolEtna\WObj:=wobjEtna;
    TriggL T2202,v50,laserON,z0,toolEtna\WObj:=wobjEtna;
    TriggL T2203,vl,laserOFF,z0,toolEtna\WObj:=wobjEtna;
    TriggL T2204,v50,laserON,z0,toolEtna\WObj:=wobjEtna;
    TriggL T2205,vl,laserOFF,z0,toolEtna\WObj:=wobjEtna;
    TriggL T2206,v50,laserON,z0,toolEtna\WObj:=wobjEtna;
    TriggL T2207,vl,laserOFF,z0,toolEtna\WObj:=wobjEtna;
    TriggL T2208,v50,laserON,z0,toolEtna\WObj:=wobjEtna;
    TriggL T2209,vl,laserOFF,z0,toolEtna\WObj:=wobjEtna;
    TriggL T2210,v50,laserON,z0,toolEtna\WObj:=wobjEtna;
    TriggL T2211,vl,laserOFF,z0,toolEtna\WObj:=wobjEtna;
    TriggL T2212,v50,laserON,z0,toolEtna\WObj:=wobjEtna;
    TriggL T2213,vl,laserOFF,z0,toolEtna\WObj:=wobjEtna;
    TriggL T2214,v50,laserON,z0,toolEtna\WObj:=wobjEtna;
    TriggL T2215,vl,laserOFF,z0,toolEtna\WObj:=wobjEtna;
    TriggL T2216,v50,laserON,z0,toolEtna\WObj:=wobjEtna;
    TriggL T2217,vl,laserOFF,z0,toolEtna\WObj:=wobjEtna;
    TriggL T2218,v50,laserON,z0,toolEtna\WObj:=wobjEtna;
    TriggL T2219,vl,laserOFF,z0,toolEtna\WObj:=wobjEtna;
    TriggL T2220,v50,laserON,z0,toolEtna\WObj:=wobjEtna;
    TriggL T2221,vl,laserOFF,z0,toolEtna\WObj:=wobjEtna;
    TriggL T2222,v50,laserON,z0,toolEtna\WObj:=wobjEtna;
    TriggL T2223,vl,laserOFF,z0,toolEtna\WObj:=wobjEtna;
    TriggL T2224,v50,laserON,z0,toolEtna\WObj:=wobjEtna;
    TriggL T2225,vl,laserOFF,z0,toolEtna\WObj:=wobjEtna;
    TriggL T2226,v50,laserON,z0,toolEtna\WObj:=wobjEtna;
    TriggL T2227,vl,laserOFF,z0,toolEtna\WObj:=wobjEtna;
    TriggL T2228,v50,laserON,z0,toolEtna\WObj:=wobjEtna;
    TriggL T2229,vl,laserOFF,z0,toolEtna\WObj:=wobjEtna;
    TriggL T2230,v50,laserON,z0,toolEtna\WObj:=wobjEtna;
    TriggL T2231,vl,laserOFF,z0,toolEtna\WObj:=wobjEtna;
    TriggL T2232,v50,laserON,z0,toolEtna\WObj:=wobjEtna;
    TriggL T2233,vl,laserOFF,z0,toolEtna\WObj:=wobjEtna;
    TriggL T2234,v50,laserON,z0,toolEtna\WObj:=wobjEtna;
    TriggL T2235,vl,laserOFF,z0,toolEtna\WObj:=wobjEtna;
    TriggL T2236,v50,laserON,z0,toolEtna\WObj:=wobjEtna;
    TriggL T2237,vl,laserOFF,z0,toolEtna\WObj:=wobjEtna;
    TriggL T2238,v50,laserON,z0,toolEtna\WObj:=wobjEtna;
    TriggL T2239,vl,laserOFF,z0,toolEtna\WObj:=wobjEtna;
    TriggL T2240,v50,laserON,z0,toolEtna\WObj:=wobjEtna;
    TriggL T2241,vl,laserOFF,z0,toolEtna\WObj:=wobjEtna;
    TriggL T2242,v50,laserON,z0,toolEtna\WObj:=wobjEtna;
    TriggL T2243,vl,laserOFF,z0,toolEtna\WObj:=wobjEtna;
    TriggL T2244,v50,laserON,z0,toolEtna\WObj:=wobjEtna;
    TriggL T2245,vl,laserOFF,z0,toolEtna\WObj:=wobjEtna;
    TriggL T2246,v50,laserON,z0,toolEtna\WObj:=wobjEtna;
    TriggL T2247,vl,laserOFF,z0,toolEtna\WObj:=wobjEtna;
    TriggL T2248,v50,laserON,z0,toolEtna\WObj:=wobjEtna;
    TriggL T2249,vl,laserOFF,z0,toolEtna\WObj:=wobjEtna;
    TriggL T2250,v50,laserON,z0,toolEtna\WObj:=wobjEtna;
    TriggL T2251,vl,laserOFF,z0,toolEtna\WObj:=wobjEtna;
    TriggL T2252,v50,laserON,z0,toolEtna\WObj:=wobjEtna;
    TriggL T2253,vl,laserOFF,z0,toolEtna\WObj:=wobjEtna;
    TriggL T2254,v50,laserON,z0,toolEtna\WObj:=wobjEtna;
    TriggL T2255,vl,laserOFF,z0,toolEtna\WObj:=wobjEtna;
    TriggL T2256,v50,laserON,z0,toolEtna\WObj:=wobjEtna;
    TriggL T2257,vl,laserOFF,z0,toolEtna\WObj:=wobjEtna;
    TriggL T2258,v50,laserON,z0,toolEtna\WObj:=wobjEtna;
    TriggL T2259,vl,laserOFF,z0,toolEtna\WObj:=wobjEtna;
    TriggL T2260,v50,laserON,z0,toolEtna\WObj:=wobjEtna;
    TriggL T2261,vl,laserOFF,z0,toolEtna\WObj:=wobjEtna;
    TriggL T2262,v50,laserON,z0,toolEtna\WObj:=wobjEtna;
    TriggL T2263,vl,laserOFF,z0,toolEtna\WObj:=wobjEtna;
    TriggL T2264,v50,laserON,z0,toolEtna\WObj:=wobjEtna;
    TriggL T2265,vl,laserOFF,z0,toolEtna\WObj:=wobjEtna;
    TriggL T2266,v50,laserON,z0,toolEtna\WObj:=wobjEtna;
    TriggL T2267,vl,laserOFF,z0,toolEtna\WObj:=wobjEtna;
    TriggL T2268,v50,laserON,z0,toolEtna\WObj:=wobjEtna;
    TriggL T2269,vl,laserOFF,z0,toolEtna\WObj:=wobjEtna;
    TriggL T2270,v50,laserON,z0,toolEtna\WObj:=wobjEtna;
    TriggL T2271,vl,laserOFF,z0,toolEtna\WObj:=wobjEtna;
    TriggL T2272,v50,laserON,z0,toolEtna\WObj:=wobjEtna;
    TriggL T2273,vl,laserOFF,z0,toolEtna\WObj:=wobjEtna;
    TriggL T2274,v50,laserON,z0,toolEtna\WObj:=wobjEtna;
    TriggL T2275,vl,laserOFF,z0,toolEtna\WObj:=wobjEtna;
    TriggL T2276,v50,laserON,z0,toolEtna\WObj:=wobjEtna;
    TriggL T2277,vl,laserOFF,z0,toolEtna\WObj:=wobjEtna;
    TriggL T2278,v50,laserON,z0,toolEtna\WObj:=wobjEtna;
    TriggL T2279,vl,laserOFF,z0,toolEtna\WObj:=wobjEtna;
    TriggL T2280,v50,laserON,z0,toolEtna\WObj:=wobjEtna;
    TriggL T2281,vl,laserOFF,z0,toolEtna\WObj:=wobjEtna;
    TriggL T2282,v50,laserON,z0,toolEtna\WObj:=wobjEtna;
    TriggL T2283,vl,laserOFF,z0,toolEtna\WObj:=wobjEtna;
    TriggL T2284,v50,laserON,z0,toolEtna\WObj:=wobjEtna;
    TriggL T2285,vl,laserOFF,z0,toolEtna\WObj:=wobjEtna;
    TriggL T2286,v50,laserON,z0,toolEtna\WObj:=wobjEtna;
    TriggL T2287,vl,laserOFF,z0,toolEtna\WObj:=wobjEtna;
    TriggL T2288,v50,laserON,z0,toolEtna\WObj:=wobjEtna;
    TriggL T2289,vl,laserOFF,z0,toolEtna\WObj:=wobjEtna;
    TriggL T2290,v50,laserON,z0,toolEtna\WObj:=wobjEtna;
    TriggL T2291,vl,laserOFF,z0,toolEtna\WObj:=wobjEtna;
    TriggL T2292,v50,laserON,z0,toolEtna\WObj:=wobjEtna;
    TriggL T2293,vl,laserOFF,z0,toolEtna\WObj:=wobjEtna;
    TriggL T2294,v50,laserON,z0,toolEtna\WObj:=wobjEtna;
    TriggL T2295,vl,laserOFF,z0,toolEtna\WObj:=wobjEtna;
    TriggL T2296,v50,laserON,z0,toolEtna\WObj:=wobjEtna;
    TriggL T2297,vl,laserOFF,z0,toolEtna\WObj:=wobjEtna;
    TriggL T2298,v50,laserON,z0,toolEtna\WObj:=wobjEtna;
    TriggL T2299,vl,laserOFF,z0,toolEtna\WObj:=wobjEtna;
    TriggL T2300,v50,laserON,z0,toolEtna\WObj:=wobjEtna;
    TriggL T2301,vl,laserOFF,z0,toolEtna\WObj:=wobjEtna;
    TriggL T2302,v50,laserON,z0,toolEtna\WObj:=wobjEtna;
    TriggL T2303,vl,laserOFF,z0,toolEtna\WObj:=wobjEtna;
    TriggL T2304,v50,laserON,z0,toolEtna\WObj:=wobjEtna;
    TriggL T2305,vl,laserOFF,z0,toolEtna\WObj:=wobjEtna;
    TriggL T2306,v50,laserON,z0,toolEtna\WObj:=wobjEtna;
    TriggL T2307,vl,laserOFF,z0,toolEtna\WObj:=wobjEtna;
    TriggL T2308,v50,laserON,z0,toolEtna\WObj:=wobjEtna;
    TriggL T2309,vl,laserOFF,z0,toolEtna\WObj:=wobjEtna;
    TriggL T2310,v50,laserON,z0,toolEtna\WObj:=wobjEtna;
    TriggL T2311,vl,laserOFF,z0,toolEtna\WObj:=wobjEtna;
    TriggL T2312,v50,laserON,z0,toolEtna\WObj:=wobjEtna;
    TriggL T2313,vl,laserOFF,z0,toolEtna\WObj:=wobjEtna;
    TriggL T2314,v50,laserON,z0,toolEtna\WObj:=wobjEtna;
    TriggL T2315,vl,laserOFF,z0,toolEtna\WObj:=wobjEtna;
    TriggL T2316,v50,laserON,z0,toolEtna\WObj:=wobjEtna;
    TriggL T2317,vl,laserOFF,z0,toolEtna\WObj:=wobjEtna;
    TriggL T2318,v50,laserON,z0,toolEtna\WObj:=wobjEtna;
    TriggL T2319,vl,laserOFF,z0,toolEtna\WObj:=wobjEtna;
    TriggL T2320,v50,laserON,z0,toolEtna\WObj:=wobjEtna;
    TriggL T2321,vl,laserOFF,z0,toolEtna\WObj:=wobjEtna;
    TriggL T2322,v50,laserON,z0,toolEtna\WObj:=wobjEtna;
    TriggL T2323,vl,laserOFF,z0,toolEtna\WObj:=wobjEtna;
    TriggL T2324,v50,laserON,z0,toolEtna\WObj:=wobjEtna;
    TriggL T2325,vl,laserOFF,z0,toolEtna\WObj:=wobjEtna;
    TriggL T2326,v50,laserON,z0,toolEtna\WObj:=wobjEtna;
    TriggL T2327,vl,laserOFF,z0,toolEtna\WObj:=wobjEtna;
    TriggL T2328,v50,laserON,z0,toolEtna\WObj:=wobjEtna;
    TriggL T2329,vl,laserOFF,z0,toolEtna\WObj:=wobjEtna;
    TriggL T2330,v50,laserON,z0,toolEtna\WObj:=wobjEtna;
    TriggL T2331,vl,laserOFF,z0,toolEtna\WObj:=wobjEtna;
    TriggL T2332,v50,laserON,z0,toolEtna\WObj:=wobjEtna;
    TriggL T2333,vl,laserOFF,z0,toolEtna\WObj:=wobjEtna;
    TriggL T2334,v50,laserON,z0,toolEtna\WObj:=wobjEtna;
    TriggL T2335,vl,laserOFF,z0,toolEtna\WObj:=wobjEtna;
    TriggL T2336,v50,laserON,z0,toolEtna\WObj:=wobjEtna;
    TriggL T2337,vl,laserOFF,z0,toolEtna\WObj:=wobjEtna;
    TriggL T2338,v50,laserON,z0,toolEtna\WObj:=wobjEtna;
    TriggL T2339,vl,laserOFF,z0,toolEtna\WObj:=wobjEtna;
    TriggL T2340,v50,laserON,z0,toolEtna\WObj:=wobjEtna;
    TriggL T2341,vl,laserOFF,z0,toolEtna\WObj:=wobjEtna;
    TriggL T2342,v50,laserON,z0,toolEtna\WObj:=wobjEtna;
    TriggL T2343,vl,laserOFF,z0,toolEtna\WObj:=wobjEtna;
    TriggL T2344,v50,laserON,z0,toolEtna\WObj:=wobjEtna;
    TriggL T2345,vl,laserOFF,z0,toolEtna\WObj:=wobjEtna;
    TriggL T2346,v50,laserON,z0,toolEtna\WObj:=wobjEtna;
    TriggL T2347,vl,laserOFF,z0,toolEtna\WObj:=wobjEtna;
    TriggL T2348,v50,laserON,z0,toolEtna\WObj:=wobjEtna;
    TriggL T2349,vl,laserOFF,z0,toolEtna\WObj:=wobjEtna;
    TriggL T2350,v50,laserON,z0,toolEtna\WObj:=wobjEtna;
    TriggL T2351,vl,laserOFF,z0,toolEtna\WObj:=wobjEtna;
    TriggL T2352,v50,laserON,z0,toolEtna\WObj:=wobjEtna;
    TriggL T2353,vl,laserOFF,z0,toolEtna\WObj:=wobjEtna;
    TriggL T2354,v50,laserON,z0,toolEtna\WObj:=wobjEtna;
    TriggL T2355,vl,laserOFF,z0,toolEtna\WObj:=wobjEtna;
    TriggL T2356,v50,laserON,z0,toolEtna\WObj:=wobjEtna;
    TriggL T2357,vl,laserOFF,z0,toolEtna\WObj:=wobjEtna;
    TriggL T2358,v50,laserON,z0,toolEtna\WObj:=wobjEtna;
    TriggL T2359,vl,laserOFF,z0,toolEtna\WObj:=wobjEtna;
    TriggL T2360,v50,laserON,z0,toolEtna\WObj:=wobjEtna;
    TriggL T2361,vl,laserOFF,z0,toolEtna\WObj:=wobjEtna;
    TriggL T2362,v50,laserON,z0,toolEtna\WObj:=wobjEtna;
    TriggL T2363,vl,laserOFF,z0,toolEtna\WObj:=wobjEtna;
    TriggL T2364,v50,laserON,z0,toolEtna\WObj:=wobjEtna;
    TriggL T2365,vl,laserOFF,z0,toolEtna\WObj:=wobjEtna;
    TriggL T2366,v50,laserON,z0,toolEtna\WObj:=wobjEtna;
    TriggL T2367,vl,laserOFF,z0,toolEtna\WObj:=wobjEtna;
    TriggL T2368,v50,laserON,z0,toolEtna\WObj:=wobjEtna;
    TriggL T2369,vl,laserOFF,z0,toolEtna\WObj:=wobjEtna;
    TriggL T2370,v50,laserON,z0,toolEtna\WObj:=wobjEtna;
    TriggL T2371,vl,laserOFF,z0,toolEtna\WObj:=wobjEtna;
    TriggL T2372,v50,laserON,z0,toolEtna\WObj:=wobjEtna;
    TriggL T2373,vl,laserOFF,z0,toolEtna\WObj:=wobjEtna;
    TriggL T2374,v50,laserON,z0,toolEtna\WObj:=wobjEtna;
    TriggL T2375,vl,laserOFF,z0,toolEtna\WObj:=wobjEtna;
    TriggL T2376,v50,laserON,z0,toolEtna\WObj:=wobjEtna;
    TriggL T2377,vl,laserOFF,z0,toolEtna\WObj:=wobjEtna;
    TriggL T2378,v50,laserON,z0,toolEtna\WObj:=wobjEtna;
    TriggL T2379,vl,laserOFF,z0,toolEtna\WObj:=wobjEtna;
    TriggL T2380,v50,laserON,z0,toolEtna\WObj:=wobjEtna;
    TriggL T2381,vl,laserOFF,z0,toolEtna\WObj:=wobjEtna;
    TriggL T2382,v50,laserON,z0,toolEtna\WObj:=wobjEtna;
    TriggL T2383,vl,laserOFF,z0,toolEtna\WObj:=wobjEtna;
    TriggL T2384,v50,laserON,z0,toolEtna\WObj:=wobjEtna;
    TriggL T2385,vl,laserOFF,z0,toolEtna\WObj:=wobjEtna;
    TriggL T2386,v50,laserON,z0,toolEtna\WObj:=wobjEtna;
    TriggL T2387,vl,laserOFF,z0,toolEtna\WObj:=wobjEtna;
    TriggL T2388,v50,laserON,z0,toolEtna\WObj:=wobjEtna;
    TriggL T2389,vl,laserOFF,z0,toolEtna\WObj:=wobjEtna;
    TriggL T2390,v50,laserON,z0,toolEtna\WObj:=wobjEtna;
    TriggL T2391,vl,laserOFF,z0,toolEtna\WObj:=wobjEtna;
    TriggL T2392,v50,laserON,z0,toolEtna\WObj:=wobjEtna;
    TriggL T2393,vl,laserOFF,z0,toolEtna\WObj:=wobjEtna;
    TriggL T2394,v50,laserON,z0,toolEtna\WObj:=wobjEtna;
    TriggL T2395,vl,laserOFF,z0,toolEtna\WObj:=wobjEtna;
    TriggL T2396,v50,laserON,z0,toolEtna\WObj:=wobjEtna;
    TriggL T2397,vl,laserOFF,z0,toolEtna\WObj:=wobjEtna;
    TriggL T2398,v50,laserON,z0,toolEtna\WObj:=wobjEtna;
    TriggL T2399,vl,laserOFF,z0,toolEtna\WObj:=wobjEtna;
    TriggL T2400,v50,laserON,z0,toolEtna\WObj:=wobjEtna;
    TriggL T2401,vl,laserOFF,z0,toolEtna\WObj:=wobjEtna;
    TriggL T2402,v50,laserON,z0,toolEtna\WObj:=wobjEtna;
    TriggL T2403,vl,laserOFF,z0,toolEtna\WObj:=wobjEtna;
    TriggL T2404,v50,laserON,z0,toolEtna\WObj:=wobjEtna;
    TriggL T2405,vl,laserOFF,z0,toolEtna\WObj:=wobjEtna;
    TriggL T2406,v50,laserON,z0,toolEtna\WObj:=wobjEtna;
    TriggL T2407,vl,laserOFF,z0,toolEtna\WObj:=wobjEtna;
    TriggL T2408,v50,laserON,z0,toolEtna\WObj:=wobjEtna;
    TriggL T2409,vl,laserOFF,z0,toolEtna\WObj:=wobjEtna;
    TriggL T2410,v50,laserON,z0,toolEtna\WObj:=wobjEtna;
    TriggL T2411,vl,laserOFF,z0,toolEtna\WObj:=wobjEtna;
    TriggL T2412,v50,laserON,z0,toolEtna\WObj:=wobjEtna;
    TriggL T2413,vl,laserOFF,z0,toolEtna\WObj:=wobjEtna;
    TriggL T2414,v50,laserON,z0,toolEtna\WObj:=wobjEtna;
    TriggL T2415,vl,laserOFF,z0,toolEtna\WObj:=wobjEtna;
    TriggL T2416,v50,laserON,z0,toolEtna\WObj:=wobjEtna;
    TriggL T2417,vl,laserOFF,z0,toolEtna\WObj:=wobjEtna;
    TriggL T2418,v50,laserON,z0,toolEtna\WObj:=wobjEtna;
    TriggL T2419,vl,laserOFF,z0,toolEtna\WObj:=wobjEtna;
    TriggL T2420,v50,laserON,z0,toolEtna\WObj:=wobjEtna;
    TriggL T2421,vl,laserOFF,z0,toolEtna\WObj:=wobjEtna;
    TriggL T2422,v50,laserON,z0,toolEtna\WObj:=wobjEtna;
    TriggL T2423,vl,laserOFF,z0,toolEtna\WObj:=wobjEtna;
    TriggL T2424,v50,laserON,z0,toolEtna\WObj:=wobjEtna;
    TriggL T2425,vl,laserOFF,z0,toolEtna\WObj:=wobjEtna;
    TriggL T2426,v50,laserON,z0,toolEtna\WObj:=wobjEtna;
    TriggL T2427,vl,laserOFF,z0,toolEtna\WObj:=wobjEtna;
    TriggL T2428,v50,laserON,z0,toolEtna\WObj:=wobjEtna;
    TriggL T2429,vl,laserOFF,z0,toolEtna\WObj:=wobjEtna;
    TriggL T2430,v50,laserON,z0,toolEtna\WObj:=wobjEtna;
    TriggL T2431,vl,laserOFF,z0,toolEtna\WObj:=wobjEtna;
    TriggL T2432,v50,laserON,z0,toolEtna\WObj:=wobjEtna;
    TriggL T2433,vl,laserOFF,z0,toolEtna\WObj:=wobjEtna;
    TriggL T2434,v50,laserON,z0,toolEtna\WObj:=wobjEtna;
    TriggL T2435,vl,laserOFF,z0,toolEtna\WObj:=wobjEtna;
    TriggL T2436,v50,laserON,z0,toolEtna\WObj:=wobjEtna;
    TriggL T2437,vl,laserOFF,z0,toolEtna\WObj:=wobjEtna;
    TriggL T2438,v50,laserON,z0,toolEtna\WObj:=wobjEtna;
    TriggL T2439,vl,laserOFF,z0,toolEtna\WObj:=wobjEtna;
    TriggL T2440,v50,laserON,z0,toolEtna\WObj:=wobjEtna;
    TriggL T2441,vl,laserOFF,z0,toolEtna\WObj:=wobjEtna;
    TriggL T2442,v50,laserON,z0,toolEtna\WObj:=wobjEtna;
    TriggL T2443,vl,laserOFF,z0,toolEtna\WObj:=wobjEtna;
    TriggL T2444,v50,laserON,z0,toolEtna\WObj:=wobjEtna;
    TriggL T2445,vl,laserOFF,z0,toolEtna\WObj:=wobjEtna;
    TriggL T2446,v50,laserON,z0,toolEtna\WObj:=wobjEtna;
    TriggL T2447,vl,laserOFF,z0,toolEtna\WObj:=wobjEtna;
    TriggL T2448,v50,laserON,z0,toolEtna\WObj:=wobjEtna;
    TriggL T2449,vl,laserOFF,z0,toolEtna\WObj:=wobjEtna;
    TriggL T2450,v50,laserON,z0,toolEtna\WObj:=wobjEtna;
    TriggL T2451,vl,laserOFF,z0,toolEtna\WObj:=wobjEtna;
    TriggL T2452,v50,laserON,z0,toolEtna\WObj:=wobjEtna;
    TriggL T2453,vl,laserOFF,z0,toolEtna\WObj:=wobjEtna;
    TriggL T2454,v50,laserON,z0,toolEtna\WObj:=wobjEtna;
    TriggL T2455,vl,laserOFF,z0,toolEtna\WObj:=wobjEtna;
    TriggL T2456,v50,laserON,z0,toolEtna\WObj:=wobjEtna;
    TriggL T2457,vl,laserOFF,z0,toolEtna\WObj:=wobjEtna;
    TriggL T2458,v50,laserON,z0,toolEtna\WObj:=wobjEtna;
    TriggL T2459,vl,laserOFF,z0,toolEtna\WObj:=wobjEtna;
    TriggL T2460,v50,laserON,z0,toolEtna\WObj:=wobjEtna;
    TriggL T2461,vl,laserOFF,z0,toolEtna\WObj:=wobjEtna;
    TriggL T2462,v50,laserON,z0,toolEtna\WObj:=wobjEtna;
    TriggL T2463,vl,laserOFF,z0,toolEtna\WObj:=wobjEtna;
    TriggL T2464,v50,laserON,z0,toolEtna\WObj:=wobjEtna;
    TriggL T2465,vl,laserOFF,z0,toolEtna\WObj:=wobjEtna;
    TriggL T2466,v50,laserON,z0,toolEtna\WObj:=wobjEtna;
    TriggL T2467,vl,laserOFF,z0,toolEtna\WObj:=wobjEtna;
    TriggL T2468,v50,laserON,z0,toolEtna\WObj:=wobjEtna;
    TriggL T2469,vl,laserOFF,z0,toolEtna\WObj:=wobjEtna;
    TriggL T2470,v50,laserON,z0,toolEtna\WObj:=wobjEtna;
    TriggL T2471,vl,laserOFF,z0,toolEtna\WObj:=wobjEtna;
    TriggL T2472,v50,laserON,z0,toolEtna\WObj:=wobjEtna;
    TriggL T2473,vl,laserOFF,z0,toolEtna\WObj:=wobjEtna;
    TriggL T2474,v50,laserON,z0,toolEtna\WObj:=wobjEtna;
    TriggL T2475,vl,laserOFF,z0,toolEtna\WObj:=wobjEtna;
    TriggL T2476,v50,laserON,z0,toolEtna\WObj:=wobjEtna;
    TriggL T2477,vl,laserOFF,z0,toolEtna\WObj:=wobjEtna;
    TriggL T2478,v50,laserON,z0,toolEtna\WObj:=wobjEtna;
    TriggL T2479,vl,laserOFF,z0,toolEtna\WObj:=wobjEtna;
    TriggL T2480,v50,laserON,z0,toolEtna\WObj:=wobjEtna;
    TriggL T2481,vl,laserOFF,z0,toolEtna\WObj:=wobjEtna;
    TriggL T2482,v50,laserON,z0,toolEtna\WObj:=wobjEtna;
    TriggL T2483,vl,laserOFF,z0,toolEtna\WObj:=wobjEtna;
    TriggL T2484,v50,laserON,z0,toolEtna\WObj:=wobjEtna;
    TriggL T2485,vl,laserOFF,z0,toolEtna\WObj:=wobjEtna;
    TriggL T2486,v50,laserON,z0,toolEtna\WObj:=wobjEtna;
    TriggL T2487,vl,laserOFF,z0,toolEtna\WObj:=wobjEtna;
    TriggL T2488,v50,laserON,z0,toolEtna\WObj:=wobjEtna;
    TriggL T2489,vl,laserOFF,z0,toolEtna\WObj:=wobjEtna;
    TriggL T2490,v50,laserON,z0,toolEtna\WObj:=wobjEtna;
    TriggL T2491,vl,laserOFF,z0,toolEtna\WObj:=wobjEtna;
    TriggL T2492,v50,laserON,z0,toolEtna\WObj:=wobjEtna;
    TriggL T2493,vl,laserOFF,z0,toolEtna\WObj:=wobjEtna;
    TriggL T2494,v50,laserON,z0,toolEtna\WObj:=wobjEtna;
    TriggL T2495,vl,laserOFF,z0,toolEtna\WObj:=wobjEtna;
    TriggL T2496,v50,laserON,z0,toolEtna\WObj:=wobjEtna;
    TriggL T2497,vl,laserOFF,z0,toolEtna\WObj:=wobjEtna;
    TriggL T2498,v50,laserON,z0,toolEtna\WObj:=wobjEtna;
    TriggL T2499,vl,laserOFF,z0,toolEtna\WObj:=wobjEtna;
    TriggL T2500,v50,laserON,z0,toolEtna\WObj:=wobjEtna;
    TriggL T2501,vl,laserOFF,z0,toolEtna\WObj:=wobjEtna;
    TriggL T2502,v50,laserON,z0,toolEtna\WObj:=wobjEtna;
    TriggL T2503,vl,laserOFF,z0,toolEtna\WObj:=wobjEtna;
    TriggL T2504,v50,laserON,z0,toolEtna\WObj:=wobjEtna;
    TriggL T2505,vl,laserOFF,z0,toolEtna\WObj:=wobjEtna;
    TriggL T2506,v50,laserON,z0,toolEtna\WObj:=wobjEtna;
    TriggL T2507,vl,laserOFF,z0,toolEtna\WObj:=wobjEtna;
    TriggL T2508,v50,laserON,z0,toolEtna\WObj:=wobjEtna;
    TriggL T2509,vl,laserOFF,z0,toolEtna\WObj:=wobjEtna;
    TriggL T2510,v50,laserON,z0,toolEtna\WObj:=wobjEtna;
    TriggL T2511,vl,laserOFF,z0,toolEtna\WObj:=wobjEtna;
    TriggL T2512,v50,laserON,z0,toolEtna\WObj:=wobjEtna;
    TriggL T2513,vl,laserOFF,z0,toolEtna\WObj:=wobjEtna;
    TriggL T2514,v50,laserON,z0,toolEtna\WObj:=wobjEtna;
    TriggL T2515,vl,laserOFF,z0,toolEtna\WObj:=wobjEtna;
    TriggL T2516,v50,laserON,z0,toolEtna\WObj:=wobjEtna;
    TriggL T2517,vl,laserOFF,z0,toolEtna\WObj:=wobjEtna;
    TriggL T2518,v50,laserON,z0,toolEtna\WObj:=wobjEtna;
    TriggL T2519,vl,laserOFF,z0,toolEtna\WObj:=wobjEtna;
    TriggL T2520,v50,laserON,z0,toolEtna\WObj:=wobjEtna;
    TriggL T2521,vl,laserOFF,z0,toolEtna\WObj:=wobjEtna;
    TriggL T2522,v50,laserON,z0,toolEtna\WObj:=wobjEtna;
    TriggL T2523,vl,laserOFF,z0,toolEtna\WObj:=wobjEtna;
    TriggL T2524,v50,laserON,z0,toolEtna\WObj:=wobjEtna;
    TriggL T2525,vl,laserOFF,z0,toolEtna\WObj:=wobjEtna;
    TriggL T2526,v50,laserON,z0,toolEtna\WObj:=wobjEtna;
    TriggL T2527,vl,laserOFF,z0,toolEtna\WObj:=wobjEtna;
    TriggL T2528,v50,laserON,z0,toolEtna\WObj:=wobjEtna;
    TriggL T2529,vl,laserOFF,z0,toolEtna\WObj:=wobjEtna;
    TriggL T2530,v50,laserON,z0,toolEtna\WObj:=wobjEtna;
    TriggL T2531,vl,laserOFF,z0,toolEtna\WObj:=wobjEtna;
    TriggL T2532,v50,laserON,z0,toolEtna\WObj:=wobjEtna;
    TriggL T2533,vl,laserOFF,z0,toolEtna\WObj:=wobjEtna;
    TriggL T2534,v50,laserON,z0,toolEtna\WObj:=wobjEtna;
    TriggL T2535,vl,laserOFF,z0,toolEtna\WObj:=wobjEtna;
    TriggL T2536,v50,laserON,z0,toolEtna\WObj:=wobjEtna;
    TriggL T2537,vl,laserOFF,z0,toolEtna\WObj:=wobjEtna;
    TriggL T2538,v50,laserON,z0,toolEtna\WObj:=wobjEtna;
    TriggL T2539,vl,laserOFF,z0,toolEtna\WObj:=wobjEtna;
    TriggL T2540,v50,laserON,z0,toolEtna\WObj:=wobjEtna;
    TriggL T2541,vl,laserOFF,z0,toolEtna\WObj:=wobjEtna;
    TriggL T2542,v50,laserON,z0,toolEtna\WObj:=wobjEtna;
    TriggL T2543,vl,laserOFF,z0,toolEtna\WObj:=wobjEtna;
    TriggL T2544,v50,laserON,z0,toolEtna\WObj:=wobjEtna;
    TriggL T2545,vl,laserOFF,z0,toolEtna\WObj:=wobjEtna;
    TriggL T2546,v50,laserON,z0,toolEtna\WObj:=wobjEtna;
    TriggL T2547,vl,laserOFF,z0,toolEtna\WObj:=wobjEtna;
    TriggL T2548,v50,laserON,z0,toolEtna\WObj:=wobjEtna;
    TriggL T2549,vl,laserOFF,z0,toolEtna\WObj:=wobjEtna;
    TriggL T2550,v50,laserON,z0,toolEtna\WObj:=wobjEtna;
    TriggL T2551,vl,laserOFF,z0,toolEtna\WObj:=wobjEtna;
    TriggL T2552,v50,laserON,z0,toolEtna\WObj:=wobjEtna;
    TriggL T2553,vl,laserOFF,z0,toolEtna\WObj:=wobjEtna;
    TriggL T2554,v50,laserON,z0,toolEtna\WObj:=wobjEtna;
    TriggL T2555,vl,laserOFF,z0,toolEtna\WObj:=wobjEtna;
    TriggL T2556,v50,laserON,z0,toolEtna\WObj:=wobjEtna;
    TriggL T2557,vl,laserOFF,z0,toolEtna\WObj:=wobjEtna;
    TriggL T2558,v50,laserON,z0,toolEtna\WObj:=wobjEtna;
    TriggL T2559,vl,laserOFF,z0,toolEtna\WObj:=wobjEtna;
    TriggL T2560,v50,laserON,z0,toolEtna\WObj:=wobjEtna;
    TriggL T2561,vl,laserOFF,z0,toolEtna\WObj:=wobjEtna;
    TriggL T2562,v50,laserON,z0,toolEtna\WObj:=wobjEtna;
    TriggL T2563,vl,laserOFF,z0,toolEtna\WObj:=wobjEtna;
    TriggL T2564,v50,laserON,z0,toolEtna\WObj:=wobjEtna;
    TriggL T2565,vl,laserOFF,z0,toolEtna\WObj:=wobjEtna;
    TriggL T2566,v50,laserON,z0,toolEtna\WObj:=wobjEtna;
    TriggL T2567,vl,laserOFF,z0,toolEtna\WObj:=wobjEtna;
    TriggL T2568,v50,laserON,z0,toolEtna\WObj:=wobjEtna;
    TriggL T2569,vl,laserOFF,z0,toolEtna\WObj:=wobjEtna;
    TriggL T2570,v50,laserON,z0,toolEtna\WObj:=wobjEtna;
    TriggL T2571,vl,laserOFF,z0,toolEtna\WObj:=wobjEtna;
    TriggL T2572,v50,laserON,z0,toolEtna\WObj:=wobjEtna;
    TriggL T2573,vl,laserOFF,z0,toolEtna\WObj:=wobjEtna;
    TriggL T2574,v50,laserON,z0,toolEtna\WObj:=wobjEtna;
    TriggL T2575,vl,laserOFF,z0,toolEtna\WObj:=wobjEtna;
    TriggL T2576,v50,laserON,z0,toolEtna\WObj:=wobjEtna;
    TriggL T2577,vl,laserOFF,z0,toolEtna\WObj:=wobjEtna;
    TriggL T2578,v50,laserON,z0,toolEtna\WObj:=wobjEtna;
    TriggL T2579,vl,laserOFF,z0,toolEtna\WObj:=wobjEtna;
    TriggL T2580,v50,laserON,z0,toolEtna\WObj:=wobjEtna;
    TriggL T2581,vl,laserOFF,z0,toolEtna\WObj:=wobjEtna;
    TriggL T2582,v50,laserON,z0,toolEtna\WObj:=wobjEtna;
    TriggL T2583,vl,laserOFF,z0,toolEtna\WObj:=wobjEtna;
    TriggL T2584,v50,laserON,z0,toolEtna\WObj:=wobjEtna;
    TriggL T2585,vl,laserOFF,z0,toolEtna\WObj:=wobjEtna;
    TriggL T2586,v50,laserON,z0,toolEtna\WObj:=wobjEtna;
    TriggL T2587,vl,laserOFF,z0,toolEtna\WObj:=wobjEtna;
    TriggL T2588,v50,laserON,z0,toolEtna\WObj:=wobjEtna;
    TriggL T2589,vl,laserOFF,z0,toolEtna\WObj:=wobjEtna;
    TriggL T2590,v50,laserON,z0,toolEtna\WObj:=wobjEtna;
    TriggL T2591,vl,laserOFF,z0,toolEtna\WObj:=wobjEtna;
    TriggL T2592,v50,laserON,z0,toolEtna\WObj:=wobjEtna;
    TriggL T2593,vl,laserOFF,z0,toolEtna\WObj:=wobjEtna;
    TriggL T2594,v50,laserON,z0,toolEtna\WObj:=wobjEtna;
    TriggL T2595,vl,laserOFF,z0,toolEtna\WObj:=wobjEtna;
    TriggL T2596,v50,laserON,z0,toolEtna\WObj:=wobjEtna;
    TriggL T2597,vl,laserOFF,z0,toolEtna\WObj:=wobjEtna;
    TriggL T2598,v50,laserON,z0,toolEtna\WObj:=wobjEtna;
    TriggL T2599,vl,laserOFF,z0,toolEtna\WObj:=wobjEtna;
    TriggL T2600,v50,laserON,z0,toolEtna\WObj:=wobjEtna;
    TriggL T2601,vl,laserOFF,z0,toolEtna\WObj:=wobjEtna;
    TriggL T2602,v50,laserON,z0,toolEtna\WObj:=wobjEtna;
    TriggL T2603,vl,laserOFF,z0,toolEtna\WObj:=wobjEtna;
    TriggL T2604,v50,laserON,z0,toolEtna\WObj:=wobjEtna;
    TriggL T2605,vl,laserOFF,z0,toolEtna\WObj:=wobjEtna;
    TriggL T2606,v50,laserON,z0,toolEtna\WObj:=wobjEtna;
    TriggL T2607,vl,laserOFF,z0,toolEtna\WObj:=wobjEtna;
    TriggL T2608,v50,laserON,z0,toolEtna\WObj:=wobjEtna;
    TriggL T2609,vl,laserOFF,z0,toolEtna\WObj:=wobjEtna;
    TriggL T2610,v50,laserON,z0,toolEtna\WObj:=wobjEtna;
    TriggL T2611,vl,laserOFF,z0,toolEtna\WObj:=wobjEtna;
    TriggL T2612,v50,laserON,z0,toolEtna\WObj:=wobjEtna;
    TriggL T2613,vl,laserOFF,z0,toolEtna\WObj:=wobjEtna;
    TriggL T2614,v50,laserON,z0,toolEtna\WObj:=wobjEtna;
    TriggL T2615,vl,laserOFF,z0,toolEtna\WObj:=wobjEtna;
    TriggL T2616,v50,laserON,z0,toolEtna\WObj:=wobjEtna;
    TriggL T2617,vl,laserOFF,z0,toolEtna\WObj:=wobjEtna;
    TriggL T2618,v50,laserON,z0,toolEtna\WObj:=wobjEtna;
    TriggL T2619,vl,laserOFF,z0,toolEtna\WObj:=wobjEtna;
    TriggL T2620,v50,laserON,z0,toolEtna\WObj:=wobjEtna;
    TriggL T2621,vl,laserOFF,z0,toolEtna\WObj:=wobjEtna;
    TriggL T2622,v50,laserON,z0,toolEtna\WObj:=wobjEtna;
    TriggL T2623,vl,laserOFF,z0,toolEtna\WObj:=wobjEtna;
    TriggL T2624,v50,laserON,z0,toolEtna\WObj:=wobjEtna;
    TriggL T2625,vl,laserOFF,z0,toolEtna\WObj:=wobjEtna;
    TriggL T2626,v50,laserON,z0,toolEtna\WObj:=wobjEtna;
    TriggL T2627,vl,laserOFF,z0,toolEtna\WObj:=wobjEtna;
    TriggL T2628,v50,laserON,z0,toolEtna\WObj:=wobjEtna;
    TriggL T2629,vl,laserOFF,z0,toolEtna\WObj:=wobjEtna;
    TriggL T2630,v50,laserON,z0,toolEtna\WObj:=wobjEtna;
    TriggL T2631,vl,laserOFF,z0,toolEtna\WObj:=wobjEtna;
    TriggL T2632,v50,laserON,z0,toolEtna\WObj:=wobjEtna;
    TriggL T2633,vl,laserOFF,z0,toolEtna\WObj:=wobjEtna;
    TriggL T2634,v50,laserON,z0,toolEtna\WObj:=wobjEtna;
    TriggL T2635,vl,laserOFF,z0,toolEtna\WObj:=wobjEtna;
    TriggL T2636,v50,laserON,z0,toolEtna\WObj:=wobjEtna;
    TriggL T2637,vl,laserOFF,z0,toolEtna\WObj:=wobjEtna;
    TriggL T2638,v50,laserON,z0,toolEtna\WObj:=wobjEtna;
    TriggL T2639,vl,laserOFF,z0,toolEtna\WObj:=wobjEtna;
    TriggL T2640,v50,laserON,z0,toolEtna\WObj:=wobjEtna;
    TriggL T2641,vl,laserOFF,z0,toolEtna\WObj:=wobjEtna;
    TriggL T2642,v50,laserON,z0,toolEtna\WObj:=wobjEtna;
    TriggL T2643,vl,laserOFF,z0,toolEtna\WObj:=wobjEtna;
    TriggL T2644,v50,laserON,z0,toolEtna\WObj:=wobjEtna;
    TriggL T2645,vl,laserOFF,z0,toolEtna\WObj:=wobjEtna;
    TriggL T2646,v50,laserON,z0,toolEtna\WObj:=wobjEtna;
    TriggL T2647,vl,laserOFF,z0,toolEtna\WObj:=wobjEtna;
    TriggL T2648,v50,laserON,z0,toolEtna\WObj:=wobjEtna;
    TriggL T2649,vl,laserOFF,z0,toolEtna\WObj:=wobjEtna;
    TriggL T2650,v50,laserON,z0,toolEtna\WObj:=wobjEtna;
    TriggL T2651,vl,laserOFF,z0,toolEtna\WObj:=wobjEtna;
    TriggL T2652,v50,laserON,z0,toolEtna\WObj:=wobjEtna;
    TriggL T2653,vl,laserOFF,z0,toolEtna\WObj:=wobjEtna;
    TriggL T2654,v50,laserON,z0,toolEtna\WObj:=wobjEtna;
    TriggL T2655,vl,laserOFF,z0,toolEtna\WObj:=wobjEtna;
    TriggL T2656,v50,laserON,z0,toolEtna\WObj:=wobjEtna;
    TriggL T2657,vl,laserOFF,z0,toolEtna\WObj:=wobjEtna;
    TriggL T2658,v50,laserON,z0,toolEtna\WObj:=wobjEtna;
    TriggL T2659,vl,laserOFF,z0,toolEtna\WObj:=wobjEtna;
    TriggL T2660,v50,laserON,z0,toolEtna\WObj:=wobjEtna;
    TriggL T2661,vl,laserOFF,z0,toolEtna\WObj:=wobjEtna;
    TriggL T2662,v50,laserON,z0,toolEtna\WObj:=wobjEtna;
    TriggL T2663,vl,laserOFF,z0,toolEtna\WObj:=wobjEtna;
    TriggL T2664,v50,laserON,z0,toolEtna\WObj:=wobjEtna;
    TriggL T2665,vl,laserOFF,z0,toolEtna\WObj:=wobjEtna;
    TriggL T2666,v50,laserON,z0,toolEtna\WObj:=wobjEtna;
    TriggL T2667,vl,laserOFF,z0,toolEtna\WObj:=wobjEtna;
    TriggL T2668,v50,laserON,z0,toolEtna\WObj:=wobjEtna;
    TriggL T2669,vl,laserOFF,z0,toolEtna\WObj:=wobjEtna;
    TriggL T2670,v50,laserON,z0,toolEtna\WObj:=wobjEtna;
    TriggL T2671,vl,laserOFF,z0,toolEtna\WObj:=wobjEtna;
    TriggL T2672,v50,laserON,z0,toolEtna\WObj:=wobjEtna;
    TriggL T2673,vl,laserOFF,z0,toolEtna\WObj:=wobjEtna;
    TriggL T2674,v50,laserON,z0,toolEtna\WObj:=wobjEtna;
    TriggL T2675,vl,laserOFF,z0,toolEtna\WObj:=wobjEtna;
    TriggL T2676,v50,laserON,z0,toolEtna\WObj:=wobjEtna;
    TriggL T2677,vl,laserOFF,z0,toolEtna\WObj:=wobjEtna;
    TriggL T2678,v50,laserON,z0,toolEtna\WObj:=wobjEtna;
    TriggL T2679,vl,laserOFF,z0,toolEtna\WObj:=wobjEtna;
    TriggL T2680,v50,laserON,z0,toolEtna\WObj:=wobjEtna;
    TriggL T2681,vl,laserOFF,z0,toolEtna\WObj:=wobjEtna;
    TriggL T2682,v50,laserON,z0,toolEtna\WObj:=wobjEtna;
    TriggL T2683,vl,laserOFF,z0,toolEtna\WObj:=wobjEtna;
    TriggL T2684,v50,laserON,z0,toolEtna\WObj:=wobjEtna;
    TriggL T2685,vl,laserOFF,z0,toolEtna\WObj:=wobjEtna;
    TriggL T2686,v50,laserON,z0,toolEtna\WObj:=wobjEtna;
    TriggL T2687,vl,laserOFF,z0,toolEtna\WObj:=wobjEtna;
    TriggL T2688,v50,laserON,z0,toolEtna\WObj:=wobjEtna;
    TriggL T2689,vl,laserOFF,z0,toolEtna\WObj:=wobjEtna;
    TriggL T2690,v50,laserON,z0,toolEtna\WObj:=wobjEtna;
    TriggL T2691,vl,laserOFF,z0,toolEtna\WObj:=wobjEtna;
    TriggL T2692,v50,laserON,z0,toolEtna\WObj:=wobjEtna;
    TriggL T2693,vl,laserOFF,z0,toolEtna\WObj:=wobjEtna;
    TriggL T2694,v50,laserON,z0,toolEtna\WObj:=wobjEtna;
    TriggL T2695,vl,laserOFF,z0,toolEtna\WObj:=wobjEtna;
    TriggL T2696,v50,laserON,z0,toolEtna\WObj:=wobjEtna;
    TriggL T2697,vl,laserOFF,z0,toolEtna\WObj:=wobjEtna;
    TriggL T2698,v50,laserON,z0,toolEtna\WObj:=wobjEtna;
    TriggL T2699,vl,laserOFF,z0,toolEtna\WObj:=wobjEtna;
    TriggL T2700,v50,laserON,z0,toolEtna\WObj:=wobjEtna;
    TriggL T2701,vl,laserOFF,z0,toolEtna\WObj:=wobjEtna;
    TriggL T2702,v50,laserON,z0,toolEtna\WObj:=wobjEtna;
    TriggL T2703,vl,laserOFF,z0,toolEtna\WObj:=wobjEtna;
    TriggL T2704,v50,laserON,z0,toolEtna\WObj:=wobjEtna;
    TriggL T2705,vl,laserOFF,z0,toolEtna\WObj:=wobjEtna;
    TriggL T2706,v50,laserON,z0,toolEtna\WObj:=wobjEtna;
    TriggL T2707,vl,laserOFF,z0,toolEtna\WObj:=wobjEtna;
    TriggL T2708,v50,laserON,z0,toolEtna\WObj:=wobjEtna;
    TriggL T2709,vl,laserOFF,z0,toolEtna\WObj:=wobjEtna;
    TriggL T2710,v50,laserON,z0,toolEtna\WObj:=wobjEtna;
    TriggL T2711,vl,laserOFF,z0,toolEtna\WObj:=wobjEtna;
    TriggL T2712,v50,laserON,z0,toolEtna\WObj:=wobjEtna;
    TriggL T2713,vl,laserOFF,z0,toolEtna\WObj:=wobjEtna;
    TriggL T2714,v50,laserON,z0,toolEtna\WObj:=wobjEtna;
    TriggL T2715,vl,laserOFF,z0,toolEtna\WObj:=wobjEtna;
    TriggL T2716,v50,laserON,z0,toolEtna\WObj:=wobjEtna;
    TriggL T2717,vl,laserOFF,z0,toolEtna\WObj:=wobjEtna;
    TriggL T2718,v50,laserON,z0,toolEtna\WObj:=wobjEtna;
    TriggL T2719,vl,laserOFF,z0,toolEtna\WObj:=wobjEtna;
    TriggL T2720,v50,laserON,z0,toolEtna\WObj:=wobjEtna;
    TriggL T2721,vl,laserOFF,z0,toolEtna\WObj:=wobjEtna;
    TriggL T2722,v50,laserON,z0,toolEtna\WObj:=wobjEtna;
    TriggL T2723,vl,laserOFF,z0,toolEtna\WObj:=wobjEtna;
    TriggL T2724,v50,laserON,z0,toolEtna\WObj:=wobjEtna;
    TriggL T2725,vl,laserOFF,z0,toolEtna\WObj:=wobjEtna;
    TriggL T2726,v50,laserON,z0,toolEtna\WObj:=wobjEtna;
    TriggL T2727,vl,laserOFF,z0,toolEtna\WObj:=wobjEtna;
    TriggL T2728,v50,laserON,z0,toolEtna\WObj:=wobjEtna;
    TriggL T2729,vl,laserOFF,z0,toolEtna\WObj:=wobjEtna;
    TriggL T2730,v50,laserON,z0,toolEtna\WObj:=wobjEtna;
    TriggL T2731,vl,laserOFF,z0,toolEtna\WObj:=wobjEtna;
    TriggL T2732,v50,laserON,z0,toolEtna\WObj:=wobjEtna;
    TriggL T2733,vl,laserOFF,z0,toolEtna\WObj:=wobjEtna;
    TriggL T2734,v50,laserON,z0,toolEtna\WObj:=wobjEtna;
    TriggL T2735,vl,laserOFF,z0,toolEtna\WObj:=wobjEtna;
    TriggL T2736,v50,laserON,z0,toolEtna\WObj:=wobjEtna;
    TriggL T2737,vl,laserOFF,z0,toolEtna\WObj:=wobjEtna;
    TriggL T2738,v50,laserON,z0,toolEtna\WObj:=wobjEtna;
    TriggL T2739,vl,laserOFF,z0,toolEtna\WObj:=wobjEtna;
    TriggL T2740,v50,laserON,z0,toolEtna\WObj:=wobjEtna;
    TriggL T2741,vl,laserOFF,z0,toolEtna\WObj:=wobjEtna;
    TriggL T2742,v50,laserON,z0,toolEtna\WObj:=wobjEtna;
    TriggL T2743,vl,laserOFF,z0,toolEtna\WObj:=wobjEtna;
    TriggL T2744,v50,laserON,z0,toolEtna\WObj:=wobjEtna;
    TriggL T2745,vl,laserOFF,z0,toolEtna\WObj:=wobjEtna;
    TriggL T2746,v50,laserON,z0,toolEtna\WObj:=wobjEtna;
    TriggL T2747,vl,laserOFF,z0,toolEtna\WObj:=wobjEtna;
    TriggL T2748,v50,laserON,z0,toolEtna\WObj:=wobjEtna;
    TriggL T2749,vl,laserOFF,z0,toolEtna\WObj:=wobjEtna;
    TriggL T2750,v50,laserON,z0,toolEtna\WObj:=wobjEtna;
    TriggL T2751,vl,laserOFF,z0,toolEtna\WObj:=wobjEtna;
    TriggL T2752,v50,laserON,z0,toolEtna\WObj:=wobjEtna;
    TriggL T2753,vl,laserOFF,z0,toolEtna\WObj:=wobjEtna;
    TriggL T2754,v50,laserON,z0,toolEtna\WObj:=wobjEtna;
    TriggL T2755,vl,laserOFF,z0,toolEtna\WObj:=wobjEtna;
    TriggL T2756,v50,laserON,z0,toolEtna\WObj:=wobjEtna;
    TriggL T2757,vl,laserOFF,z0,toolEtna\WObj:=wobjEtna;
    TriggL T2758,v50,laserON,z0,toolEtna\WObj:=wobjEtna;
    TriggL T2759,vl,laserOFF,z0,toolEtna\WObj:=wobjEtna;
    TriggL T2760,v50,laserON,z0,toolEtna\WObj:=wobjEtna;
    TriggL T2761,vl,laserOFF,z0,toolEtna\WObj:=wobjEtna;
    TriggL T2762,v50,laserON,z0,toolEtna\WObj:=wobjEtna;
    TriggL T2763,vl,laserOFF,z0,toolEtna\WObj:=wobjEtna;
    TriggL T2764,v50,laserON,z0,toolEtna\WObj:=wobjEtna;
    TriggL T2765,vl,laserOFF,z0,toolEtna\WObj:=wobjEtna;
    TriggL T2766,v50,laserON,z0,toolEtna\WObj:=wobjEtna;
    TriggL T2767,vl,laserOFF,z0,toolEtna\WObj:=wobjEtna;
    TriggL T2768,v50,laserON,z0,toolEtna\WObj:=wobjEtna;
    TriggL T2769,vl,laserOFF,z0,toolEtna\WObj:=wobjEtna;
    TriggL T2770,v50,laserON,z0,toolEtna\WObj:=wobjEtna;
    TriggL T2771,vl,laserOFF,z0,toolEtna\WObj:=wobjEtna;
    TriggL T2772,v50,laserON,z0,toolEtna\WObj:=wobjEtna;
    TriggL T2773,vl,laserOFF,z0,toolEtna\WObj:=wobjEtna;
    TriggL T2774,v50,laserON,z0,toolEtna\WObj:=wobjEtna;
    TriggL T2775,vl,laserOFF,z0,toolEtna\WObj:=wobjEtna;
    TriggL T2776,v50,laserON,z0,toolEtna\WObj:=wobjEtna;
    TriggL T2777,vl,laserOFF,z0,toolEtna\WObj:=wobjEtna;
    TriggL T2778,v50,laserON,z0,toolEtna\WObj:=wobjEtna;
    TriggL T2779,vl,laserOFF,z0,toolEtna\WObj:=wobjEtna;
    TriggL T2780,v50,laserON,z0,toolEtna\WObj:=wobjEtna;
    TriggL T2781,vl,laserOFF,z0,toolEtna\WObj:=wobjEtna;
    TriggL T2782,v50,laserON,z0,toolEtna\WObj:=wobjEtna;
    TriggL T2783,vl,laserOFF,z0,toolEtna\WObj:=wobjEtna;
    TriggL T2784,v50,laserON,z0,toolEtna\WObj:=wobjEtna;
    TriggL T2785,vl,laserOFF,z0,toolEtna\WObj:=wobjEtna;
    TriggL T2786,v50,laserON,z0,toolEtna\WObj:=wobjEtna;
    TriggL T2787,vl,laserOFF,z0,toolEtna\WObj:=wobjEtna;
    TriggL T2788,v50,laserON,z0,toolEtna\WObj:=wobjEtna;
    TriggL T2789,vl,laserOFF,z0,toolEtna\WObj:=wobjEtna;
    TriggL T2790,v50,laserON,z0,toolEtna\WObj:=wobjEtna;
    TriggL T2791,vl,laserOFF,z0,toolEtna\WObj:=wobjEtna;
    TriggL T2792,v50,laserON,z0,toolEtna\WObj:=wobjEtna;
    TriggL T2793,vl,laserOFF,z0,toolEtna\WObj:=wobjEtna;
    TriggL T2794,v50,laserON,z0,toolEtna\WObj:=wobjEtna;
    TriggL T2795,vl,laserOFF,z0,toolEtna\WObj:=wobjEtna;
    TriggL T2796,v50,laserON,z0,toolEtna\WObj:=wobjEtna;
    TriggL T2797,vl,laserOFF,z0,toolEtna\WObj:=wobjEtna;
    TriggL T2798,v50,laserON,z0,toolEtna\WObj:=wobjEtna;
    TriggL T2799,vl,laserOFF,z0,toolEtna\WObj:=wobjEtna;
    TriggL T2800,v50,laserON,z0,toolEtna\WObj:=wobjEtna;
    TriggL T2801,vl,laserOFF,z0,toolEtna\WObj:=wobjEtna;
    TriggL T2802,v50,laserON,z0,toolEtna\WObj:=wobjEtna;
    TriggL T2803,vl,laserOFF,z0,toolEtna\WObj:=wobjEtna;
    TriggL T2804,v50,laserON,z0,toolEtna\WObj:=wobjEtna;
    TriggL T2805,vl,laserOFF,z0,toolEtna\WObj:=wobjEtna;
    TriggL T2806,v50,laserON,z0,toolEtna\WObj:=wobjEtna;
    TriggL T2807,vl,laserOFF,z0,toolEtna\WObj:=wobjEtna;
    TriggL T2808,v50,laserON,z0,toolEtna\WObj:=wobjEtna;
    TriggL T2809,vl,laserOFF,z0,toolEtna\WObj:=wobjEtna;
    TriggL T2810,v50,laserON,z0,toolEtna\WObj:=wobjEtna;
    TriggL T2811,vl,laserOFF,z0,toolEtna\WObj:=wobjEtna;
    TriggL T2812,v50,laserON,z0,toolEtna\WObj:=wobjEtna;
    TriggL T2813,vl,laserOFF,z0,toolEtna\WObj:=wobjEtna;
    TriggL T2814,v50,laserON,z0,toolEtna\WObj:=wobjEtna;
    TriggL T2815,vl,laserOFF,z0,toolEtna\WObj:=wobjEtna;
    TriggL T2816,v50,laserON,z0,toolEtna\WObj:=wobjEtna;
    TriggL T2817,vl,laserOFF,z0,toolEtna\WObj:=wobjEtna;
    TriggL T2818,v50,laserON,z0,toolEtna\WObj:=wobjEtna;
    TriggL T2819,vl,laserOFF,z0,toolEtna\WObj:=wobjEtna;
    TriggL T2820,v50,laserON,z0,toolEtna\WObj:=wobjEtna;
    TriggL T2821,vl,laserOFF,z0,toolEtna\WObj:=wobjEtna;
    TriggL T2822,v50,laserON,z0,toolEtna\WObj:=wobjEtna;
    TriggL T2823,vl,laserOFF,z0,toolEtna\WObj:=wobjEtna;
    TriggL T2824,v50,laserON,z0,toolEtna\WObj:=wobjEtna;
    TriggL T2825,vl,laserOFF,z0,toolEtna\WObj:=wobjEtna;
    TriggL T2826,v50,laserON,z0,toolEtna\WObj:=wobjEtna;
    TriggL T2827,vl,laserOFF,z0,toolEtna\WObj:=wobjEtna;
    TriggL T2828,v50,laserON,z0,toolEtna\WObj:=wobjEtna;
    TriggL T2829,vl,laserOFF,z0,toolEtna\WObj:=wobjEtna;
    TriggL T2830,v50,laserON,z0,toolEtna\WObj:=wobjEtna;
    TriggL T2831,vl,laserOFF,z0,toolEtna\WObj:=wobjEtna;
    TriggL T2832,v50,laserON,z0,toolEtna\WObj:=wobjEtna;
    TriggL T2833,vl,laserOFF,z0,toolEtna\WObj:=wobjEtna;
    TriggL T2834,v50,laserON,z0,toolEtna\WObj:=wobjEtna;
    TriggL T2835,vl,laserOFF,z0,toolEtna\WObj:=wobjEtna;
    TriggL T2836,v50,laserON,z0,toolEtna\WObj:=wobjEtna;
    TriggL T2837,vl,laserOFF,z0,toolEtna\WObj:=wobjEtna;
    TriggL T2838,v50,laserON,z0,toolEtna\WObj:=wobjEtna;
    TriggL T2839,vl,laserOFF,z0,toolEtna\WObj:=wobjEtna;
    TriggL T2840,v50,laserON,z0,toolEtna\WObj:=wobjEtna;
    TriggL T2841,vl,laserOFF,z0,toolEtna\WObj:=wobjEtna;
    TriggL T2842,v50,laserON,z0,toolEtna\WObj:=wobjEtna;
    TriggL T2843,vl,laserOFF,z0,toolEtna\WObj:=wobjEtna;
    TriggL T2844,v50,laserON,z0,toolEtna\WObj:=wobjEtna;
    TriggL T2845,vl,laserOFF,z0,toolEtna\WObj:=wobjEtna;
    TriggL T2846,v50,laserON,z0,toolEtna\WObj:=wobjEtna;
    TriggL T2847,vl,laserOFF,z0,toolEtna\WObj:=wobjEtna;
    TriggL T2848,v50,laserON,z0,toolEtna\WObj:=wobjEtna;
    TriggL T2849,vl,laserOFF,z0,toolEtna\WObj:=wobjEtna;
    TriggL T2850,v50,laserON,z0,toolEtna\WObj:=wobjEtna;
    TriggL T2851,vl,laserOFF,z0,toolEtna\WObj:=wobjEtna;
    TriggL T2852,v50,laserON,z0,toolEtna\WObj:=wobjEtna;
    TriggL T2853,vl,laserOFF,z0,toolEtna\WObj:=wobjEtna;
    TriggL T2854,v50,laserON,z0,toolEtna\WObj:=wobjEtna;
    TriggL T2855,vl,laserOFF,z0,toolEtna\WObj:=wobjEtna;
    TriggL T2856,v50,laserON,z0,toolEtna\WObj:=wobjEtna;
    TriggL T2857,vl,laserOFF,z0,toolEtna\WObj:=wobjEtna;
    TriggL T2858,v50,laserON,z0,toolEtna\WObj:=wobjEtna;
    TriggL T2859,vl,laserOFF,z0,toolEtna\WObj:=wobjEtna;
    TriggL T2860,v50,laserON,z0,toolEtna\WObj:=wobjEtna;
    TriggL T2861,vl,laserOFF,z0,toolEtna\WObj:=wobjEtna;
    TriggL T2862,v50,laserON,z0,toolEtna\WObj:=wobjEtna;
    TriggL T2863,vl,laserOFF,z0,toolEtna\WObj:=wobjEtna;
    TriggL T2864,v50,laserON,z0,toolEtna\WObj:=wobjEtna;
    TriggL T2865,vl,laserOFF,z0,toolEtna\WObj:=wobjEtna;
    TriggL T2866,v50,laserON,z0,toolEtna\WObj:=wobjEtna;
    TriggL T2867,vl,laserOFF,z0,toolEtna\WObj:=wobjEtna;
    TriggL T2868,v50,laserON,z0,toolEtna\WObj:=wobjEtna;
    TriggL T2869,vl,laserOFF,z0,toolEtna\WObj:=wobjEtna;
    TriggL T2870,v50,laserON,z0,toolEtna\WObj:=wobjEtna;
    TriggL T2871,vl,laserOFF,z0,toolEtna\WObj:=wobjEtna;
    TriggL T2872,v50,laserON,z0,toolEtna\WObj:=wobjEtna;
    TriggL T2873,vl,laserOFF,z0,toolEtna\WObj:=wobjEtna;
    TriggL T2874,v50,laserON,z0,toolEtna\WObj:=wobjEtna;
    TriggL T2875,vl,laserOFF,z0,toolEtna\WObj:=wobjEtna;
    TriggL T2876,v50,laserON,z0,toolEtna\WObj:=wobjEtna;
    TriggL T2877,vl,laserOFF,z0,toolEtna\WObj:=wobjEtna;
    TriggL T2878,v50,laserON,z0,toolEtna\WObj:=wobjEtna;
    TriggL T2879,vl,laserOFF,z0,toolEtna\WObj:=wobjEtna;
    TriggL T2880,v50,laserON,z0,toolEtna\WObj:=wobjEtna;
    TriggL T2881,vl,laserOFF,z0,toolEtna\WObj:=wobjEtna;
    TriggL T2882,v50,laserON,z0,toolEtna\WObj:=wobjEtna;
    TriggL T2883,vl,laserOFF,z0,toolEtna\WObj:=wobjEtna;
    TriggL T2884,v50,laserON,z0,toolEtna\WObj:=wobjEtna;
    TriggL T2885,vl,laserOFF,z0,toolEtna\WObj:=wobjEtna;
    TriggL T2886,v50,laserON,z0,toolEtna\WObj:=wobjEtna;
    TriggL T2887,vl,laserOFF,z0,toolEtna\WObj:=wobjEtna;
    TriggL T2888,v50,laserON,z0,toolEtna\WObj:=wobjEtna;
    TriggL T2889,vl,laserOFF,z0,toolEtna\WObj:=wobjEtna;
    TriggL T2890,v50,laserON,z0,toolEtna\WObj:=wobjEtna;
    TriggL T2891,vl,laserOFF,z0,toolEtna\WObj:=wobjEtna;
    TriggL T2892,v50,laserON,z0,toolEtna\WObj:=wobjEtna;
    TriggL T2893,vl,laserOFF,z0,toolEtna\WObj:=wobjEtna;
    TriggL T2894,v50,laserON,z0,toolEtna\WObj:=wobjEtna;
    TriggL T2895,vl,laserOFF,z0,toolEtna\WObj:=wobjEtna;
    TriggL T2896,v50,laserON,z0,toolEtna\WObj:=wobjEtna;
    TriggL T2897,vl,laserOFF,z0,toolEtna\WObj:=wobjEtna;
    TriggL T2898,v50,laserON,z0,toolEtna\WObj:=wobjEtna;
    TriggL T2899,vl,laserOFF,z0,toolEtna\WObj:=wobjEtna;
    TriggL T2900,v50,laserON,z0,toolEtna\WObj:=wobjEtna;
    TriggL T2901,vl,laserOFF,z0,toolEtna\WObj:=wobjEtna;
    TriggL T2902,v50,laserON,z0,toolEtna\WObj:=wobjEtna;
    TriggL T2903,vl,laserOFF,z0,toolEtna\WObj:=wobjEtna;
    TriggL T2904,v50,laserON,z0,toolEtna\WObj:=wobjEtna;
    TriggL T2905,vl,laserOFF,z0,toolEtna\WObj:=wobjEtna;
    TriggL T2906,v50,laserON,z0,toolEtna\WObj:=wobjEtna;
    TriggL T2907,vl,laserOFF,z0,toolEtna\WObj:=wobjEtna;
    TriggL T2908,v50,laserON,z0,toolEtna\WObj:=wobjEtna;
    TriggL T2909,vl,laserOFF,z0,toolEtna\WObj:=wobjEtna;
    TriggL T2910,v50,laserON,z0,toolEtna\WObj:=wobjEtna;
    TriggL T2911,vl,laserOFF,z0,toolEtna\WObj:=wobjEtna;
    TriggL T2912,v50,laserON,z0,toolEtna\WObj:=wobjEtna;
    TriggL T2913,vl,laserOFF,z0,toolEtna\WObj:=wobjEtna;
    TriggL T2914,v50,laserON,z0,toolEtna\WObj:=wobjEtna;
    TriggL T2915,vl,laserOFF,z0,toolEtna\WObj:=wobjEtna;
    TriggL T2916,v50,laserON,z0,toolEtna\WObj:=wobjEtna;
    TriggL T2917,vl,laserOFF,z0,toolEtna\WObj:=wobjEtna;
    TriggL T2918,v50,laserON,z0,toolEtna\WObj:=wobjEtna;
    TriggL T2919,vl,laserOFF,z0,toolEtna\WObj:=wobjEtna;
    TriggL T2920,v50,laserON,z0,toolEtna\WObj:=wobjEtna;
    TriggL T2921,vl,laserOFF,z0,toolEtna\WObj:=wobjEtna;
    TriggL T2922,v50,laserON,z0,toolEtna\WObj:=wobjEtna;
    TriggL T2923,vl,laserOFF,z0,toolEtna\WObj:=wobjEtna;
    TriggL T2924,v50,laserON,z0,toolEtna\WObj:=wobjEtna;
    TriggL T2925,vl,laserOFF,z0,toolEtna\WObj:=wobjEtna;
    TriggL T2926,v50,laserON,z0,toolEtna\WObj:=wobjEtna;
    TriggL T2927,vl,laserOFF,z0,toolEtna\WObj:=wobjEtna;
    TriggL T2928,v50,laserON,z0,toolEtna\WObj:=wobjEtna;
    TriggL T2929,vl,laserOFF,z0,toolEtna\WObj:=wobjEtna;
    TriggL T2930,v50,laserON,z0,toolEtna\WObj:=wobjEtna;
    TriggL T2931,vl,laserOFF,z0,toolEtna\WObj:=wobjEtna;
    TriggL T2932,v50,laserON,z0,toolEtna\WObj:=wobjEtna;
    TriggL T2933,vl,laserOFF,z0,toolEtna\WObj:=wobjEtna;
    TriggL T2934,v50,laserON,z0,toolEtna\WObj:=wobjEtna;
    TriggL T2935,vl,laserOFF,z0,toolEtna\WObj:=wobjEtna;
    TriggL T2936,v50,laserON,z0,toolEtna\WObj:=wobjEtna;
    TriggL T2937,vl,laserOFF,z0,toolEtna\WObj:=wobjEtna;
    TriggL T2938,v50,laserON,z0,toolEtna\WObj:=wobjEtna;
    TriggL T2939,vl,laserOFF,z0,toolEtna\WObj:=wobjEtna;
    TriggL T2940,v50,laserON,z0,toolEtna\WObj:=wobjEtna;
    TriggL T2941,vl,laserOFF,z0,toolEtna\WObj:=wobjEtna;
    TriggL T2942,v50,laserON,z0,toolEtna\WObj:=wobjEtna;
    TriggL T2943,vl,laserOFF,z0,toolEtna\WObj:=wobjEtna;
    TriggL T2944,v50,laserON,z0,toolEtna\WObj:=wobjEtna;
    TriggL T2945,vl,laserOFF,z0,toolEtna\WObj:=wobjEtna;
    TriggL T2946,v50,laserON,z0,toolEtna\WObj:=wobjEtna;
    TriggL T2947,vl,laserOFF,z0,toolEtna\WObj:=wobjEtna;
    TriggL T2948,v50,laserON,z0,toolEtna\WObj:=wobjEtna;
    TriggL T2949,vl,laserOFF,z0,toolEtna\WObj:=wobjEtna;
    TriggL T2950,v50,laserON,z0,toolEtna\WObj:=wobjEtna;
    TriggL T2951,vl,laserOFF,z0,toolEtna\WObj:=wobjEtna;
    TriggL T2952,v50,laserON,z0,toolEtna\WObj:=wobjEtna;
    TriggL T2953,vl,laserOFF,z0,toolEtna\WObj:=wobjEtna;
    TriggL T2954,v50,laserON,z0,toolEtna\WObj:=wobjEtna;
    TriggL T2955,vl,laserOFF,z0,toolEtna\WObj:=wobjEtna;
    TriggL T2956,v50,laserON,z0,toolEtna\WObj:=wobjEtna;
    TriggL T2957,vl,laserOFF,z0,toolEtna\WObj:=wobjEtna;
    TriggL T2958,v50,laserON,z0,toolEtna\WObj:=wobjEtna;
    TriggL T2959,vl,laserOFF,z0,toolEtna\WObj:=wobjEtna;
    TriggL T2960,v50,laserON,z0,toolEtna\WObj:=wobjEtna;
    TriggL T2961,vl,laserOFF,z0,toolEtna\WObj:=wobjEtna;
    TriggL T2962,v50,laserON,z0,toolEtna\WObj:=wobjEtna;
    TriggL T2963,vl,laserOFF,z0,toolEtna\WObj:=wobjEtna;
    TriggL T2964,v50,laserON,z0,toolEtna\WObj:=wobjEtna;
    TriggL T2965,vl,laserOFF,z0,toolEtna\WObj:=wobjEtna;
    TriggL T2966,v50,laserON,z0,toolEtna\WObj:=wobjEtna;
    TriggL T2967,vl,laserOFF,z0,toolEtna\WObj:=wobjEtna;
    TriggL T2968,v50,laserON,z0,toolEtna\WObj:=wobjEtna;
    TriggL T2969,vl,laserOFF,z0,toolEtna\WObj:=wobjEtna;
    TriggL T2970,v50,laserON,z0,toolEtna\WObj:=wobjEtna;
    TriggL T2971,vl,laserOFF,z0,toolEtna\WObj:=wobjEtna;
    TriggL T2972,v50,laserON,z0,toolEtna\WObj:=wobjEtna;
    TriggL T2973,vl,laserOFF,z0,toolEtna\WObj:=wobjEtna;
    TriggL T2974,v50,laserON,z0,toolEtna\WObj:=wobjEtna;
    TriggL T2975,vl,laserOFF,z0,toolEtna\WObj:=wobjEtna;
    TriggL T2976,v50,laserON,z0,toolEtna\WObj:=wobjEtna;
    TriggL T2977,vl,laserOFF,z0,toolEtna\WObj:=wobjEtna;
    TriggL T2978,v50,laserON,z0,toolEtna\WObj:=wobjEtna;
    TriggL T2979,vl,laserOFF,z0,toolEtna\WObj:=wobjEtna;
    TriggL T2980,v50,laserON,z0,toolEtna\WObj:=wobjEtna;
    TriggL T2981,vl,laserOFF,z0,toolEtna\WObj:=wobjEtna;
    TriggL T2982,v50,laserON,z0,toolEtna\WObj:=wobjEtna;
    TriggL T2983,vl,laserOFF,z0,toolEtna\WObj:=wobjEtna;
    TriggL T2984,v50,laserON,z0,toolEtna\WObj:=wobjEtna;
    TriggL T2985,vl,laserOFF,z0,toolEtna\WObj:=wobjEtna;
    TriggL T2986,v50,laserON,z0,toolEtna\WObj:=wobjEtna;
    TriggL T2987,vl,laserOFF,z0,toolEtna\WObj:=wobjEtna;
    TriggL T2988,v50,laserON,z0,toolEtna\WObj:=wobjEtna;
    TriggL T2989,vl,laserOFF,z0,toolEtna\WObj:=wobjEtna;
    TriggL T2990,v50,laserON,z0,toolEtna\WObj:=wobjEtna;
    TriggL T2991,vl,laserOFF,z0,toolEtna\WObj:=wobjEtna;
    TriggL T2992,v50,laserON,z0,toolEtna\WObj:=wobjEtna;
    TriggL T2993,vl,laserOFF,z0,toolEtna\WObj:=wobjEtna;
    TriggL T2994,v50,laserON,z0,toolEtna\WObj:=wobjEtna;
    TriggL T2995,vl,laserOFF,z0,toolEtna\WObj:=wobjEtna;
    TriggL T2996,v50,laserON,z0,toolEtna\WObj:=wobjEtna;
    TriggL T2997,vl,laserOFF,z0,toolEtna\WObj:=wobjEtna;
    TriggL T2998,v50,laserON,z0,toolEtna\WObj:=wobjEtna;
    TriggL T2999,vl,laserOFF,z0,toolEtna\WObj:=wobjEtna;
    TriggL T3000,v50,laserON,z0,toolEtna\WObj:=wobjEtna;
    TriggL T3001,vl,laserOFF,z0,toolEtna\WObj:=wobjEtna;
    TriggL T3002,v50,laserON,z0,toolEtna\WObj:=wobjEtna;
    TriggL T3003,vl,laserOFF,z0,toolEtna\WObj:=wobjEtna;
    TriggL T3004,v50,laserON,z0,toolEtna\WObj:=wobjEtna;
    TriggL T3005,vl,laserOFF,z0,toolEtna\WObj:=wobjEtna;
    TriggL T3006,v50,laserON,z0,toolEtna\WObj:=wobjEtna;
    TriggL T3007,vl,laserOFF,z0,toolEtna\WObj:=wobjEtna;
    TriggL T3008,v50,laserON,z0,toolEtna\WObj:=wobjEtna;
    TriggL T3009,vl,laserOFF,z0,toolEtna\WObj:=wobjEtna;
    TriggL T3010,v50,laserON,z0,toolEtna\WObj:=wobjEtna;
    TriggL T3011,vl,laserOFF,z0,toolEtna\WObj:=wobjEtna;
    TriggL T3012,v50,laserON,z0,toolEtna\WObj:=wobjEtna;
    TriggL T3013,vl,laserOFF,z0,toolEtna\WObj:=wobjEtna;
    TriggL T3014,v50,laserON,z0,toolEtna\WObj:=wobjEtna;
    TriggL T3015,vl,laserOFF,z0,toolEtna\WObj:=wobjEtna;
    TriggL T3016,v50,laserON,z0,toolEtna\WObj:=wobjEtna;
    TriggL T3017,vl,laserOFF,z0,toolEtna\WObj:=wobjEtna;
    TriggL T3018,v50,laserON,z0,toolEtna\WObj:=wobjEtna;
    TriggL T3019,vl,laserOFF,z0,toolEtna\WObj:=wobjEtna;
    TriggL T3020,v50,laserON,z0,toolEtna\WObj:=wobjEtna;
    TriggL T3021,vl,laserOFF,z0,toolEtna\WObj:=wobjEtna;
    TriggL T3022,v50,laserON,z0,toolEtna\WObj:=wobjEtna;
    TriggL T3023,vl,laserOFF,z0,toolEtna\WObj:=wobjEtna;
    TriggL T3024,v50,laserON,z0,toolEtna\WObj:=wobjEtna;
    TriggL T3025,vl,laserOFF,z0,toolEtna\WObj:=wobjEtna;
    TriggL T3026,v50,laserON,z0,toolEtna\WObj:=wobjEtna;
    TriggL T3027,vl,laserOFF,z0,toolEtna\WObj:=wobjEtna;
    TriggL T3028,v50,laserON,z0,toolEtna\WObj:=wobjEtna;
    TriggL T3029,vl,laserOFF,z0,toolEtna\WObj:=wobjEtna;
    TriggL T3030,v50,laserON,z0,toolEtna\WObj:=wobjEtna;
    TriggL T3031,vl,laserOFF,z0,toolEtna\WObj:=wobjEtna;
    TriggL T3032,v50,laserON,z0,toolEtna\WObj:=wobjEtna;
    TriggL T3033,vl,laserOFF,z0,toolEtna\WObj:=wobjEtna;
    TriggL T3034,v50,laserON,z0,toolEtna\WObj:=wobjEtna;
    TriggL T3035,vl,laserOFF,z0,toolEtna\WObj:=wobjEtna;
    TriggL T3036,v50,laserON,z0,toolEtna\WObj:=wobjEtna;
    TriggL T3037,vl,laserOFF,z0,toolEtna\WObj:=wobjEtna;
    TriggL T3038,v50,laserON,z0,toolEtna\WObj:=wobjEtna;
    TriggL T3039,vl,laserOFF,z0,toolEtna\WObj:=wobjEtna;
    TriggL T3040,v50,laserON,z0,toolEtna\WObj:=wobjEtna;
    TriggL T3041,vl,laserOFF,z0,toolEtna\WObj:=wobjEtna;
    TriggL T3042,v50,laserON,z0,toolEtna\WObj:=wobjEtna;
    TriggL T3043,vl,laserOFF,z0,toolEtna\WObj:=wobjEtna;
    TriggL T3044,v50,laserON,z0,toolEtna\WObj:=wobjEtna;
    TriggL T3045,vl,laserOFF,z0,toolEtna\WObj:=wobjEtna;
    TriggL T3046,v50,laserON,z0,toolEtna\WObj:=wobjEtna;
    TriggL T3047,vl,laserOFF,z0,toolEtna\WObj:=wobjEtna;
    TriggL T3048,v50,laserON,z0,toolEtna\WObj:=wobjEtna;
    TriggL T3049,vl,laserOFF,z0,toolEtna\WObj:=wobjEtna;
    TriggL T3050,v50,laserON,z0,toolEtna\WObj:=wobjEtna;
    TriggL T3051,vl,laserOFF,z0,toolEtna\WObj:=wobjEtna;
    TriggL T3052,v50,laserON,z0,toolEtna\WObj:=wobjEtna;
    TriggL T3053,vl,laserOFF,z0,toolEtna\WObj:=wobjEtna;
    TriggL T3054,v50,laserON,z0,toolEtna\WObj:=wobjEtna;
    TriggL T3055,vl,laserOFF,z0,toolEtna\WObj:=wobjEtna;
    TriggL T3056,v50,laserON,z0,toolEtna\WObj:=wobjEtna;
    TriggL T3057,vl,laserOFF,z0,toolEtna\WObj:=wobjEtna;
    TriggL T3058,v50,laserON,z0,toolEtna\WObj:=wobjEtna;
    TriggL T3059,vl,laserOFF,z0,toolEtna\WObj:=wobjEtna;
    TriggL T3060,v50,laserON,z0,toolEtna\WObj:=wobjEtna;
    TriggL T3061,vl,laserOFF,z0,toolEtna\WObj:=wobjEtna;
    TriggL T3062,v50,laserON,z0,toolEtna\WObj:=wobjEtna;
    TriggL T3063,vl,laserOFF,z0,toolEtna\WObj:=wobjEtna;
    TriggL T3064,v50,laserON,z0,toolEtna\WObj:=wobjEtna;
    TriggL T3065,vl,laserOFF,z0,toolEtna\WObj:=wobjEtna;
    TriggL T3066,v50,laserON,z0,toolEtna\WObj:=wobjEtna;
    TriggL T3067,vl,laserOFF,z0,toolEtna\WObj:=wobjEtna;
    TriggL T3068,v50,laserON,z0,toolEtna\WObj:=wobjEtna;
    TriggL T3069,vl,laserOFF,z0,toolEtna\WObj:=wobjEtna;
    TriggL T3070,v50,laserON,z0,toolEtna\WObj:=wobjEtna;
    TriggL T3071,vl,laserOFF,z0,toolEtna\WObj:=wobjEtna;
    TriggL T3072,v50,laserON,z0,toolEtna\WObj:=wobjEtna;
    TriggL T3073,vl,laserOFF,z0,toolEtna\WObj:=wobjEtna;
    TriggL T3074,v50,laserON,z0,toolEtna\WObj:=wobjEtna;
    TriggL T3075,vl,laserOFF,z0,toolEtna\WObj:=wobjEtna;
    TriggL T3076,v50,laserON,z0,toolEtna\WObj:=wobjEtna;
    TriggL T3077,vl,laserOFF,z0,toolEtna\WObj:=wobjEtna;
    TriggL T3078,v50,laserON,z0,toolEtna\WObj:=wobjEtna;
    TriggL T3079,vl,laserOFF,z0,toolEtna\WObj:=wobjEtna;
    TriggL T3080,v50,laserON,z0,toolEtna\WObj:=wobjEtna;
    TriggL T3081,vl,laserOFF,z0,toolEtna\WObj:=wobjEtna;
    TriggL T3082,v50,laserON,z0,toolEtna\WObj:=wobjEtna;
    TriggL T3083,vl,laserOFF,z0,toolEtna\WObj:=wobjEtna;
    TriggL T3084,v50,laserON,z0,toolEtna\WObj:=wobjEtna;
    TriggL T3085,vl,laserOFF,z0,toolEtna\WObj:=wobjEtna;
    TriggL T3086,v50,laserON,z0,toolEtna\WObj:=wobjEtna;
    TriggL T3087,vl,laserOFF,z0,toolEtna\WObj:=wobjEtna;
    TriggL T3088,v50,laserON,z0,toolEtna\WObj:=wobjEtna;
    TriggL T3089,vl,laserOFF,z0,toolEtna\WObj:=wobjEtna;
    TriggL T3090,v50,laserON,z0,toolEtna\WObj:=wobjEtna;
    TriggL T3091,vl,laserOFF,z0,toolEtna\WObj:=wobjEtna;
    TriggL T3092,v50,laserON,z0,toolEtna\WObj:=wobjEtna;
    TriggL T3093,vl,laserOFF,z0,toolEtna\WObj:=wobjEtna;
    TriggL T3094,v50,laserON,z0,toolEtna\WObj:=wobjEtna;
    TriggL T3095,vl,laserOFF,z0,toolEtna\WObj:=wobjEtna;
    TriggL T3096,v50,laserON,z0,toolEtna\WObj:=wobjEtna;
    TriggL T3097,vl,laserOFF,z0,toolEtna\WObj:=wobjEtna;
    TriggL T3098,v50,laserON,z0,toolEtna\WObj:=wobjEtna;
    TriggL T3099,vl,laserOFF,z0,toolEtna\WObj:=wobjEtna;
    TriggL T3100,v50,laserON,z0,toolEtna\WObj:=wobjEtna;
    TriggL T3101,vl,laserOFF,z0,toolEtna\WObj:=wobjEtna;
    TriggL T3102,v50,laserON,z0,toolEtna\WObj:=wobjEtna;
    TriggL T3103,vl,laserOFF,z0,toolEtna\WObj:=wobjEtna;
    TriggL T3104,v50,laserON,z0,toolEtna\WObj:=wobjEtna;
    TriggL T3105,vl,laserOFF,z0,toolEtna\WObj:=wobjEtna;
    TriggL T3106,v50,laserON,z0,toolEtna\WObj:=wobjEtna;
    TriggL T3107,vl,laserOFF,z0,toolEtna\WObj:=wobjEtna;
    TriggL T3108,v50,laserON,z0,toolEtna\WObj:=wobjEtna;
    TriggL T3109,vl,laserOFF,z0,toolEtna\WObj:=wobjEtna;
    TriggL T3110,v50,laserON,z0,toolEtna\WObj:=wobjEtna;
    TriggL T3111,vl,laserOFF,z0,toolEtna\WObj:=wobjEtna;
    TriggL T3112,v50,laserON,z0,toolEtna\WObj:=wobjEtna;
    TriggL T3113,vl,laserOFF,z0,toolEtna\WObj:=wobjEtna;
    TriggL T3114,v50,laserON,z0,toolEtna\WObj:=wobjEtna;
    TriggL T3115,vl,laserOFF,z0,toolEtna\WObj:=wobjEtna;
    TriggL T3116,v50,laserON,z0,toolEtna\WObj:=wobjEtna;
    TriggL T3117,vl,laserOFF,z0,toolEtna\WObj:=wobjEtna;
    TriggL T3118,v50,laserON,z0,toolEtna\WObj:=wobjEtna;
    TriggL T3119,vl,laserOFF,z0,toolEtna\WObj:=wobjEtna;
    TriggL T3120,v50,laserON,z0,toolEtna\WObj:=wobjEtna;
    TriggL T3121,vl,laserOFF,z0,toolEtna\WObj:=wobjEtna;
    TriggL T3122,v50,laserON,z0,toolEtna\WObj:=wobjEtna;
    TriggL T3123,vl,laserOFF,z0,toolEtna\WObj:=wobjEtna;
    TriggL T3124,v50,laserON,z0,toolEtna\WObj:=wobjEtna;
    TriggL T3125,vl,laserOFF,z0,toolEtna\WObj:=wobjEtna;
    TriggL T3126,v50,laserON,z0,toolEtna\WObj:=wobjEtna;
    TriggL T3127,vl,laserOFF,z0,toolEtna\WObj:=wobjEtna;
    TriggL T3128,v50,laserON,z0,toolEtna\WObj:=wobjEtna;
    TriggL T3129,vl,laserOFF,z0,toolEtna\WObj:=wobjEtna;
    TriggL T3130,v50,laserON,z0,toolEtna\WObj:=wobjEtna;
    TriggL T3131,vl,laserOFF,z0,toolEtna\WObj:=wobjEtna;
    TriggL T3132,v50,laserON,z0,toolEtna\WObj:=wobjEtna;
    TriggL T3133,vl,laserOFF,z0,toolEtna\WObj:=wobjEtna;
    TriggL T3134,v50,laserON,z0,toolEtna\WObj:=wobjEtna;
    TriggL T3135,vl,laserOFF,z0,toolEtna\WObj:=wobjEtna;
    TriggL T3136,v50,laserON,z0,toolEtna\WObj:=wobjEtna;
    TriggL T3137,vl,laserOFF,z0,toolEtna\WObj:=wobjEtna;
    TriggL T3138,v50,laserON,z0,toolEtna\WObj:=wobjEtna;
    TriggL T3139,vl,laserOFF,z0,toolEtna\WObj:=wobjEtna;
    TriggL T3140,v50,laserON,z0,toolEtna\WObj:=wobjEtna;
    TriggL T3141,vl,laserOFF,z0,toolEtna\WObj:=wobjEtna;
    TriggL T3142,v50,laserON,z0,toolEtna\WObj:=wobjEtna;
    TriggL T3143,vl,laserOFF,z0,toolEtna\WObj:=wobjEtna;
    TriggL T3144,v50,laserON,z0,toolEtna\WObj:=wobjEtna;
    TriggL T3145,vl,laserOFF,z0,toolEtna\WObj:=wobjEtna;
    TriggL T3146,v50,laserON,z0,toolEtna\WObj:=wobjEtna;
    TriggL T3147,vl,laserOFF,z0,toolEtna\WObj:=wobjEtna;
    TriggL T3148,v50,laserON,z0,toolEtna\WObj:=wobjEtna;
    TriggL T3149,vl,laserOFF,z0,toolEtna\WObj:=wobjEtna;
    TriggL T3150,v50,laserON,z0,toolEtna\WObj:=wobjEtna;
    TriggL T3151,vl,laserOFF,z0,toolEtna\WObj:=wobjEtna;
    TriggL T3152,v50,laserON,z0,toolEtna\WObj:=wobjEtna;
    TriggL T3153,vl,laserOFF,z0,toolEtna\WObj:=wobjEtna;
    TriggL T3154,v50,laserON,z0,toolEtna\WObj:=wobjEtna;
    TriggL T3155,vl,laserOFF,z0,toolEtna\WObj:=wobjEtna;
    TriggL T3156,v50,laserON,z0,toolEtna\WObj:=wobjEtna;
    TriggL T3157,vl,laserOFF,z0,toolEtna\WObj:=wobjEtna;
    TriggL T3158,v50,laserON,z0,toolEtna\WObj:=wobjEtna;
    TriggL T3159,vl,laserOFF,z0,toolEtna\WObj:=wobjEtna;
    TriggL T3160,v50,laserON,z0,toolEtna\WObj:=wobjEtna;
    TriggL T3161,vl,laserOFF,z0,toolEtna\WObj:=wobjEtna;
    TriggL T3162,v50,laserON,z0,toolEtna\WObj:=wobjEtna;
    TriggL T3163,vl,laserOFF,z0,toolEtna\WObj:=wobjEtna;
    TriggL T3164,v50,laserON,z0,toolEtna\WObj:=wobjEtna;
    TriggL T3165,vl,laserOFF,z0,toolEtna\WObj:=wobjEtna;
    TriggL T3166,v50,laserON,z0,toolEtna\WObj:=wobjEtna;
    TriggL T3167,vl,laserOFF,z0,toolEtna\WObj:=wobjEtna;
    TriggL T3168,v50,laserON,z0,toolEtna\WObj:=wobjEtna;
    TriggL T3169,vl,laserOFF,z0,toolEtna\WObj:=wobjEtna;
    TriggL T3170,v50,laserON,z0,toolEtna\WObj:=wobjEtna;
    TriggL T3171,vl,laserOFF,z0,toolEtna\WObj:=wobjEtna;
    TriggL T3172,v50,laserON,z0,toolEtna\WObj:=wobjEtna;
    TriggL T3173,vl,laserOFF,z0,toolEtna\WObj:=wobjEtna;
    TriggL T3174,v50,laserON,z0,toolEtna\WObj:=wobjEtna;
    TriggL T3175,vl,laserOFF,z0,toolEtna\WObj:=wobjEtna;
    TriggL T3176,v50,laserON,z0,toolEtna\WObj:=wobjEtna;
    TriggL T3177,vl,laserOFF,z0,toolEtna\WObj:=wobjEtna;
    TriggL T3178,v50,laserON,z0,toolEtna\WObj:=wobjEtna;
    TriggL T3179,vl,laserOFF,z0,toolEtna\WObj:=wobjEtna;
    TriggL T3180,v50,laserON,z0,toolEtna\WObj:=wobjEtna;
    TriggL T3181,vl,laserOFF,z0,toolEtna\WObj:=wobjEtna;
    TriggL T3182,v50,laserON,z0,toolEtna\WObj:=wobjEtna;
    TriggL T3183,vl,laserOFF,z0,toolEtna\WObj:=wobjEtna;
    TriggL T3184,v50,laserON,z0,toolEtna\WObj:=wobjEtna;
    TriggL T3185,vl,laserOFF,z0,toolEtna\WObj:=wobjEtna;
    TriggL T3186,v50,laserON,z0,toolEtna\WObj:=wobjEtna;
    TriggL T3187,vl,laserOFF,z0,toolEtna\WObj:=wobjEtna;
    TriggL T3188,v50,laserON,z0,toolEtna\WObj:=wobjEtna;
    TriggL T3189,vl,laserOFF,z0,toolEtna\WObj:=wobjEtna;
    TriggL T3190,v50,laserON,z0,toolEtna\WObj:=wobjEtna;
    TriggL T3191,vl,laserOFF,z0,toolEtna\WObj:=wobjEtna;
    TriggL T3192,v50,laserON,z0,toolEtna\WObj:=wobjEtna;
    TriggL T3193,vl,laserOFF,z0,toolEtna\WObj:=wobjEtna;
    TriggL T3194,v50,laserON,z0,toolEtna\WObj:=wobjEtna;
    TriggL T3195,vl,laserOFF,z0,toolEtna\WObj:=wobjEtna;
    TriggL T3196,v50,laserON,z0,toolEtna\WObj:=wobjEtna;
    TriggL T3197,vl,laserOFF,z0,toolEtna\WObj:=wobjEtna;
    TriggL T3198,v50,laserON,z0,toolEtna\WObj:=wobjEtna;
    TriggL T3199,vl,laserOFF,z0,toolEtna\WObj:=wobjEtna;
    TriggL T3200,v50,laserON,z0,toolEtna\WObj:=wobjEtna;
    TriggL T3201,vl,laserOFF,z0,toolEtna\WObj:=wobjEtna;
    TriggL T3202,v50,laserON,z0,toolEtna\WObj:=wobjEtna;
    TriggL T3203,vl,laserOFF,z0,toolEtna\WObj:=wobjEtna;
    TriggL T3204,v50,laserON,z0,toolEtna\WObj:=wobjEtna;
    TriggL T3205,vl,laserOFF,z0,toolEtna\WObj:=wobjEtna;
    TriggL T3206,v50,laserON,z0,toolEtna\WObj:=wobjEtna;
    TriggL T3207,vl,laserOFF,z0,toolEtna\WObj:=wobjEtna;
    TriggL T3208,v50,laserON,z0,toolEtna\WObj:=wobjEtna;
    TriggL T3209,vl,laserOFF,z0,toolEtna\WObj:=wobjEtna;
    TriggL T3210,v50,laserON,z0,toolEtna\WObj:=wobjEtna;
    TriggL T3211,vl,laserOFF,z0,toolEtna\WObj:=wobjEtna;
    TriggL T3212,v50,laserON,z0,toolEtna\WObj:=wobjEtna;
    TriggL T3213,vl,laserOFF,z0,toolEtna\WObj:=wobjEtna;
    TriggL T3214,v50,laserON,z0,toolEtna\WObj:=wobjEtna;
    TriggL T3215,vl,laserOFF,z0,toolEtna\WObj:=wobjEtna;
    TriggL T3216,v50,laserON,z0,toolEtna\WObj:=wobjEtna;
    TriggL T3217,vl,laserOFF,z0,toolEtna\WObj:=wobjEtna;
    TriggL T3218,v50,laserON,z0,toolEtna\WObj:=wobjEtna;
    TriggL T3219,vl,laserOFF,z0,toolEtna\WObj:=wobjEtna;
    TriggL T3220,v50,laserON,z0,toolEtna\WObj:=wobjEtna;
    TriggL T3221,vl,laserOFF,z0,toolEtna\WObj:=wobjEtna;
    TriggL T3222,v50,laserON,z0,toolEtna\WObj:=wobjEtna;
    TriggL T3223,vl,laserOFF,z0,toolEtna\WObj:=wobjEtna;
    TriggL T3224,v50,laserON,z0,toolEtna\WObj:=wobjEtna;
    TriggL T3225,vl,laserOFF,z0,toolEtna\WObj:=wobjEtna;
    TriggL T3226,v50,laserON,z0,toolEtna\WObj:=wobjEtna;
    TriggL T3227,vl,laserOFF,z0,toolEtna\WObj:=wobjEtna;
    TriggL T3228,v50,laserON,z0,toolEtna\WObj:=wobjEtna;
    TriggL T3229,vl,laserOFF,z0,toolEtna\WObj:=wobjEtna;
    TriggL T3230,v50,laserON,z0,toolEtna\WObj:=wobjEtna;
    TriggL T3231,vl,laserOFF,z0,toolEtna\WObj:=wobjEtna;
    TriggL T3232,v50,laserON,z0,toolEtna\WObj:=wobjEtna;
    TriggL T3233,vl,laserOFF,z0,toolEtna\WObj:=wobjEtna;
    TriggL T3234,v50,laserON,z0,toolEtna\WObj:=wobjEtna;
    TriggL T3235,vl,laserOFF,z0,toolEtna\WObj:=wobjEtna;
    TriggL T3236,v50,laserON,z0,toolEtna\WObj:=wobjEtna;
    TriggL T3237,vl,laserOFF,z0,toolEtna\WObj:=wobjEtna;
    TriggL T3238,v50,laserON,z0,toolEtna\WObj:=wobjEtna;
    TriggL T3239,vl,laserOFF,z0,toolEtna\WObj:=wobjEtna;
    TriggL T3240,v50,laserON,z0,toolEtna\WObj:=wobjEtna;
    TriggL T3241,vl,laserOFF,z0,toolEtna\WObj:=wobjEtna;
    TriggL T3242,v50,laserON,z0,toolEtna\WObj:=wobjEtna;
    TriggL T3243,vl,laserOFF,z0,toolEtna\WObj:=wobjEtna;
    TriggL T3244,v50,laserON,z0,toolEtna\WObj:=wobjEtna;
    TriggL T3245,vl,laserOFF,z0,toolEtna\WObj:=wobjEtna;
    TriggL T3246,v50,laserON,z0,toolEtna\WObj:=wobjEtna;
    TriggL T3247,vl,laserOFF,z0,toolEtna\WObj:=wobjEtna;
    TriggL T3248,v50,laserON,z0,toolEtna\WObj:=wobjEtna;
    TriggL T3249,vl,laserOFF,z0,toolEtna\WObj:=wobjEtna;
    TriggL T3250,v50,laserON,z0,toolEtna\WObj:=wobjEtna;
    TriggL T3251,vl,laserOFF,z0,toolEtna\WObj:=wobjEtna;
    TriggL T3252,v50,laserON,z0,toolEtna\WObj:=wobjEtna;
    TriggL T3253,vl,laserOFF,z0,toolEtna\WObj:=wobjEtna;
    TriggL T3254,v50,laserON,z0,toolEtna\WObj:=wobjEtna;
    TriggL T3255,vl,laserOFF,z0,toolEtna\WObj:=wobjEtna;
    TriggL T3256,v50,laserON,z0,toolEtna\WObj:=wobjEtna;
    TriggL T3257,vl,laserOFF,z0,toolEtna\WObj:=wobjEtna;
    TriggL T3258,v50,laserON,z0,toolEtna\WObj:=wobjEtna;
    TriggL T3259,vl,laserOFF,z0,toolEtna\WObj:=wobjEtna;
    TriggL T3260,v50,laserON,z0,toolEtna\WObj:=wobjEtna;
    TriggL T3261,vl,laserOFF,z0,toolEtna\WObj:=wobjEtna;
    TriggL T3262,v50,laserON,z0,toolEtna\WObj:=wobjEtna;
    TriggL T3263,vl,laserOFF,z0,toolEtna\WObj:=wobjEtna;
    TriggL T3264,v50,laserON,z0,toolEtna\WObj:=wobjEtna;
    TriggL T3265,vl,laserOFF,z0,toolEtna\WObj:=wobjEtna;
    TriggL T3266,v50,laserON,z0,toolEtna\WObj:=wobjEtna;
    TriggL T3267,vl,laserOFF,z0,toolEtna\WObj:=wobjEtna;
    TriggL T3268,v50,laserON,z0,toolEtna\WObj:=wobjEtna;
    TriggL T3269,vl,laserOFF,z0,toolEtna\WObj:=wobjEtna;
    TriggL T3270,v50,laserON,z0,toolEtna\WObj:=wobjEtna;
    TriggL T3271,vl,laserOFF,z0,toolEtna\WObj:=wobjEtna;
    TriggL T3272,v50,laserON,z0,toolEtna\WObj:=wobjEtna;
    TriggL T3273,vl,laserOFF,z0,toolEtna\WObj:=wobjEtna;
    TriggL T3274,v50,laserON,z0,toolEtna\WObj:=wobjEtna;
    TriggL T3275,vl,laserOFF,z0,toolEtna\WObj:=wobjEtna;
    TriggL T3276,v50,laserON,z0,toolEtna\WObj:=wobjEtna;
    TriggL T3277,vl,laserOFF,z0,toolEtna\WObj:=wobjEtna;
    TriggL T3278,v50,laserON,z0,toolEtna\WObj:=wobjEtna;
    TriggL T3279,vl,laserOFF,z0,toolEtna\WObj:=wobjEtna;
    TriggL T3280,v50,laserON,z0,toolEtna\WObj:=wobjEtna;
    TriggL T3281,vl,laserOFF,z0,toolEtna\WObj:=wobjEtna;
    TriggL T3282,v50,laserON,z0,toolEtna\WObj:=wobjEtna;
    TriggL T3283,vl,laserOFF,z0,toolEtna\WObj:=wobjEtna;
    TriggL T3284,v50,laserON,z0,toolEtna\WObj:=wobjEtna;
    TriggL T3285,vl,laserOFF,z0,toolEtna\WObj:=wobjEtna;
    TriggL T3286,v50,laserON,z0,toolEtna\WObj:=wobjEtna;
    TriggL T3287,vl,laserOFF,z0,toolEtna\WObj:=wobjEtna;
    TriggL T3288,v50,laserON,z0,toolEtna\WObj:=wobjEtna;
    TriggL T3289,vl,laserOFF,z0,toolEtna\WObj:=wobjEtna;
    TriggL T3290,v50,laserON,z0,toolEtna\WObj:=wobjEtna;
    TriggL T3291,vl,laserOFF,z0,toolEtna\WObj:=wobjEtna;
    TriggL T3292,v50,laserON,z0,toolEtna\WObj:=wobjEtna;
    TriggL T3293,vl,laserOFF,z0,toolEtna\WObj:=wobjEtna;
    TriggL T3294,v50,laserON,z0,toolEtna\WObj:=wobjEtna;
    TriggL T3295,vl,laserOFF,z0,toolEtna\WObj:=wobjEtna;
    TriggL T3296,v50,laserON,z0,toolEtna\WObj:=wobjEtna;
    TriggL T3297,vl,laserOFF,z0,toolEtna\WObj:=wobjEtna;
    TriggL T3298,v50,laserON,z0,toolEtna\WObj:=wobjEtna;
    TriggL T3299,vl,laserOFF,z0,toolEtna\WObj:=wobjEtna;
    TriggL T3300,v50,laserON,z0,toolEtna\WObj:=wobjEtna;
    TriggL T3301,vl,laserOFF,z0,toolEtna\WObj:=wobjEtna;
    TriggL T3302,v50,laserON,z0,toolEtna\WObj:=wobjEtna;
    TriggL T3303,vl,laserOFF,z0,toolEtna\WObj:=wobjEtna;
    TriggL T3304,v50,laserON,z0,toolEtna\WObj:=wobjEtna;
    TriggL T3305,vl,laserOFF,z0,toolEtna\WObj:=wobjEtna;
    TriggL T3306,v50,laserON,z0,toolEtna\WObj:=wobjEtna;
    TriggL T3307,vl,laserOFF,z0,toolEtna\WObj:=wobjEtna;
    TriggL T3308,v50,laserON,z0,toolEtna\WObj:=wobjEtna;
    TriggL T3309,vl,laserOFF,z0,toolEtna\WObj:=wobjEtna;
    TriggL T3310,v50,laserON,z0,toolEtna\WObj:=wobjEtna;
    TriggL T3311,vl,laserOFF,z0,toolEtna\WObj:=wobjEtna;
    TriggL T3312,v50,laserON,z0,toolEtna\WObj:=wobjEtna;
    TriggL T3313,vl,laserOFF,z0,toolEtna\WObj:=wobjEtna;
    TriggL T3314,v50,laserON,z0,toolEtna\WObj:=wobjEtna;
    TriggL T3315,vl,laserOFF,z0,toolEtna\WObj:=wobjEtna;
    TriggL T3316,v50,laserON,z0,toolEtna\WObj:=wobjEtna;
    TriggL T3317,vl,laserOFF,z0,toolEtna\WObj:=wobjEtna;
    TriggL T3318,v50,laserON,z0,toolEtna\WObj:=wobjEtna;
    TriggL T3319,vl,laserOFF,z0,toolEtna\WObj:=wobjEtna;
    TriggL T3320,v50,laserON,z0,toolEtna\WObj:=wobjEtna;
    TriggL T3321,vl,laserOFF,z0,toolEtna\WObj:=wobjEtna;
    TriggL T3322,v50,laserON,z0,toolEtna\WObj:=wobjEtna;
    TriggL T3323,vl,laserOFF,z0,toolEtna\WObj:=wobjEtna;
    TriggL T3324,v50,laserON,z0,toolEtna\WObj:=wobjEtna;
    TriggL T3325,vl,laserOFF,z0,toolEtna\WObj:=wobjEtna;
    TriggL T3326,v50,laserON,z0,toolEtna\WObj:=wobjEtna;
    TriggL T3327,vl,laserOFF,z0,toolEtna\WObj:=wobjEtna;
    TriggL T3328,v50,laserON,z0,toolEtna\WObj:=wobjEtna;
    TriggL T3329,vl,laserOFF,z0,toolEtna\WObj:=wobjEtna;
    TriggL T3330,v50,laserON,z0,toolEtna\WObj:=wobjEtna;
    TriggL T3331,vl,laserOFF,z0,toolEtna\WObj:=wobjEtna;
    TriggL T3332,v50,laserON,z0,toolEtna\WObj:=wobjEtna;
    TriggL T3333,vl,laserOFF,z0,toolEtna\WObj:=wobjEtna;
    TriggL T3334,v50,laserON,z0,toolEtna\WObj:=wobjEtna;
    TriggL T3335,vl,laserOFF,z0,toolEtna\WObj:=wobjEtna;
    TriggL T3336,v50,laserON,z0,toolEtna\WObj:=wobjEtna;
    TriggL T3337,vl,laserOFF,z0,toolEtna\WObj:=wobjEtna;
    TriggL T3338,v50,laserON,z0,toolEtna\WObj:=wobjEtna;
    TriggL T3339,vl,laserOFF,z0,toolEtna\WObj:=wobjEtna;
    TriggL T3340,v50,laserON,z0,toolEtna\WObj:=wobjEtna;
    TriggL T3341,vl,laserOFF,z0,toolEtna\WObj:=wobjEtna;
    TriggL T3342,v50,laserON,z0,toolEtna\WObj:=wobjEtna;
    TriggL T3343,vl,laserOFF,z0,toolEtna\WObj:=wobjEtna;
    TriggL T3344,v50,laserON,z0,toolEtna\WObj:=wobjEtna;
    TriggL T3345,vl,laserOFF,z0,toolEtna\WObj:=wobjEtna;
    TriggL T3346,v50,laserON,z0,toolEtna\WObj:=wobjEtna;
    TriggL T3347,vl,laserOFF,z0,toolEtna\WObj:=wobjEtna;
    TriggL T3348,v50,laserON,z0,toolEtna\WObj:=wobjEtna;
    TriggL T3349,vl,laserOFF,z0,toolEtna\WObj:=wobjEtna;
    TriggL T3350,v50,laserON,z0,toolEtna\WObj:=wobjEtna;
    TriggL T3351,vl,laserOFF,z0,toolEtna\WObj:=wobjEtna;
    TriggL T3352,v50,laserON,z0,toolEtna\WObj:=wobjEtna;
    TriggL T3353,vl,laserOFF,z0,toolEtna\WObj:=wobjEtna;
    TriggL T3354,v50,laserON,z0,toolEtna\WObj:=wobjEtna;
    TriggL T3355,vl,laserOFF,z0,toolEtna\WObj:=wobjEtna;
    TriggL T3356,v50,laserON,z0,toolEtna\WObj:=wobjEtna;
    TriggL T3357,vl,laserOFF,z0,toolEtna\WObj:=wobjEtna;
    TriggL T3358,v50,laserON,z0,toolEtna\WObj:=wobjEtna;
    TriggL T3359,vl,laserOFF,z0,toolEtna\WObj:=wobjEtna;
    TriggL T3360,v50,laserON,z0,toolEtna\WObj:=wobjEtna;
    TriggL T3361,vl,laserOFF,z0,toolEtna\WObj:=wobjEtna;
    TriggL T3362,v50,laserON,z0,toolEtna\WObj:=wobjEtna;
    TriggL T3363,vl,laserOFF,z0,toolEtna\WObj:=wobjEtna;
    TriggL T3364,v50,laserON,z0,toolEtna\WObj:=wobjEtna;
    TriggL T3365,vl,laserOFF,z0,toolEtna\WObj:=wobjEtna;
    TriggL T3366,v50,laserON,z0,toolEtna\WObj:=wobjEtna;
    TriggL T3367,vl,laserOFF,z0,toolEtna\WObj:=wobjEtna;
    TriggL T3368,v50,laserON,z0,toolEtna\WObj:=wobjEtna;
    TriggL T3369,vl,laserOFF,z0,toolEtna\WObj:=wobjEtna;
    TriggL T3370,v50,laserON,z0,toolEtna\WObj:=wobjEtna;
    TriggL T3371,vl,laserOFF,z0,toolEtna\WObj:=wobjEtna;
    TriggL T3372,v50,laserON,z0,toolEtna\WObj:=wobjEtna;
    TriggL T3373,vl,laserOFF,z0,toolEtna\WObj:=wobjEtna;
    TriggL T3374,v50,laserON,z0,toolEtna\WObj:=wobjEtna;
    TriggL T3375,vl,laserOFF,z0,toolEtna\WObj:=wobjEtna;
    TriggL T3376,v50,laserON,z0,toolEtna\WObj:=wobjEtna;
    TriggL T3377,vl,laserOFF,z0,toolEtna\WObj:=wobjEtna;
    TriggL T3378,v50,laserON,z0,toolEtna\WObj:=wobjEtna;
    TriggL T3379,vl,laserOFF,z0,toolEtna\WObj:=wobjEtna;
    TriggL T3380,v50,laserON,z0,toolEtna\WObj:=wobjEtna;
    TriggL T3381,vl,laserOFF,z0,toolEtna\WObj:=wobjEtna;
    TriggL T3382,v50,laserON,z0,toolEtna\WObj:=wobjEtna;
    TriggL T3383,vl,laserOFF,z0,toolEtna\WObj:=wobjEtna;
    TriggL T3384,v50,laserON,z0,toolEtna\WObj:=wobjEtna;
    TriggL T3385,vl,laserOFF,z0,toolEtna\WObj:=wobjEtna;
    TriggL T3386,v50,laserON,z0,toolEtna\WObj:=wobjEtna;
    TriggL T3387,vl,laserOFF,z0,toolEtna\WObj:=wobjEtna;
    TriggL T3388,v50,laserON,z0,toolEtna\WObj:=wobjEtna;
    TriggL T3389,vl,laserOFF,z0,toolEtna\WObj:=wobjEtna;
    TriggL T3390,v50,laserON,z0,toolEtna\WObj:=wobjEtna;
    TriggL T3391,vl,laserOFF,z0,toolEtna\WObj:=wobjEtna;
    TriggL T3392,v50,laserON,z0,toolEtna\WObj:=wobjEtna;
    TriggL T3393,vl,laserOFF,z0,toolEtna\WObj:=wobjEtna;
    TriggL T3394,v50,laserON,z0,toolEtna\WObj:=wobjEtna;
    TriggL T3395,vl,laserOFF,z0,toolEtna\WObj:=wobjEtna;
    TriggL T3396,v50,laserON,z0,toolEtna\WObj:=wobjEtna;
    TriggL T3397,vl,laserOFF,z0,toolEtna\WObj:=wobjEtna;
    TriggL T3398,v50,laserON,z0,toolEtna\WObj:=wobjEtna;
    TriggL T3399,vl,laserOFF,z0,toolEtna\WObj:=wobjEtna;
    TriggL T3400,v50,laserON,z0,toolEtna\WObj:=wobjEtna;
    TriggL T3401,vl,laserOFF,z0,toolEtna\WObj:=wobjEtna;
    TriggL T3402,v50,laserON,z0,toolEtna\WObj:=wobjEtna;
    TriggL T3403,vl,laserOFF,z0,toolEtna\WObj:=wobjEtna;
    TriggL T3404,v50,laserON,z0,toolEtna\WObj:=wobjEtna;
    TriggL T3405,vl,laserOFF,z0,toolEtna\WObj:=wobjEtna;
    TriggL T3406,v50,laserON,z0,toolEtna\WObj:=wobjEtna;
    TriggL T3407,vl,laserOFF,z0,toolEtna\WObj:=wobjEtna;
    TriggL T3408,v50,laserON,z0,toolEtna\WObj:=wobjEtna;
    TriggL T3409,vl,laserOFF,z0,toolEtna\WObj:=wobjEtna;
    TriggL T3410,v50,laserON,z0,toolEtna\WObj:=wobjEtna;
    TriggL T3411,vl,laserOFF,z0,toolEtna\WObj:=wobjEtna;
    TriggL T3412,v50,laserON,z0,toolEtna\WObj:=wobjEtna;
    TriggL T3413,vl,laserOFF,z0,toolEtna\WObj:=wobjEtna;
    TriggL T3414,v50,laserON,z0,toolEtna\WObj:=wobjEtna;
    TriggL T3415,vl,laserOFF,z0,toolEtna\WObj:=wobjEtna;
    TriggL T3416,v50,laserON,z0,toolEtna\WObj:=wobjEtna;
    TriggL T3417,vl,laserOFF,z0,toolEtna\WObj:=wobjEtna;
    TriggL T3418,v50,laserON,z0,toolEtna\WObj:=wobjEtna;
    TriggL T3419,vl,laserOFF,z0,toolEtna\WObj:=wobjEtna;
    TriggL T3420,v50,laserON,z0,toolEtna\WObj:=wobjEtna;
    TriggL T3421,vl,laserOFF,z0,toolEtna\WObj:=wobjEtna;
    TriggL T3422,v50,laserON,z0,toolEtna\WObj:=wobjEtna;
    TriggL T3423,vl,laserOFF,z0,toolEtna\WObj:=wobjEtna;
    TriggL T3424,v50,laserON,z0,toolEtna\WObj:=wobjEtna;
    TriggL T3425,vl,laserOFF,z0,toolEtna\WObj:=wobjEtna;
    TriggL T3426,v50,laserON,z0,toolEtna\WObj:=wobjEtna;
    TriggL T3427,vl,laserOFF,z0,toolEtna\WObj:=wobjEtna;
    TriggL T3428,v50,laserON,z0,toolEtna\WObj:=wobjEtna;
    TriggL T3429,vl,laserOFF,z0,toolEtna\WObj:=wobjEtna;
    TriggL T3430,v50,laserON,z0,toolEtna\WObj:=wobjEtna;
    TriggL T3431,vl,laserOFF,z0,toolEtna\WObj:=wobjEtna;
    TriggL T3432,v50,laserON,z0,toolEtna\WObj:=wobjEtna;
    TriggL T3433,vl,laserOFF,z0,toolEtna\WObj:=wobjEtna;
    TriggL T3434,v50,laserON,z0,toolEtna\WObj:=wobjEtna;
    TriggL T3435,vl,laserOFF,z0,toolEtna\WObj:=wobjEtna;
    TriggL T3436,v50,laserON,z0,toolEtna\WObj:=wobjEtna;
    TriggL T3437,vl,laserOFF,z0,toolEtna\WObj:=wobjEtna;
    TriggL T3438,v50,laserON,z0,toolEtna\WObj:=wobjEtna;
    TriggL T3439,vl,laserOFF,z0,toolEtna\WObj:=wobjEtna;
    TriggL T3440,v50,laserON,z0,toolEtna\WObj:=wobjEtna;
    TriggL T3441,vl,laserOFF,z0,toolEtna\WObj:=wobjEtna;
    TriggL T3442,v50,laserON,z0,toolEtna\WObj:=wobjEtna;
    TriggL T3443,vl,laserOFF,z0,toolEtna\WObj:=wobjEtna;
    TriggL T3444,v50,laserON,z0,toolEtna\WObj:=wobjEtna;
    TriggL T3445,vl,laserOFF,z0,toolEtna\WObj:=wobjEtna;
    TriggL T3446,v50,laserON,z0,toolEtna\WObj:=wobjEtna;
    TriggL T3447,vl,laserOFF,z0,toolEtna\WObj:=wobjEtna;
    TriggL T3448,v50,laserON,z0,toolEtna\WObj:=wobjEtna;
    TriggL T3449,vl,laserOFF,z0,toolEtna\WObj:=wobjEtna;
    TriggL T3450,v50,laserON,z0,toolEtna\WObj:=wobjEtna;
    TriggL T3451,vl,laserOFF,z0,toolEtna\WObj:=wobjEtna;
    TriggL T3452,v50,laserON,z0,toolEtna\WObj:=wobjEtna;
    TriggL T3453,vl,laserOFF,z0,toolEtna\WObj:=wobjEtna;
    TriggL T3454,v50,laserON,z0,toolEtna\WObj:=wobjEtna;
    TriggL T3455,vl,laserOFF,z0,toolEtna\WObj:=wobjEtna;
    TriggL T3456,v50,laserON,z0,toolEtna\WObj:=wobjEtna;
    TriggL T3457,vl,laserOFF,z0,toolEtna\WObj:=wobjEtna;
    TriggL T3458,v50,laserON,z0,toolEtna\WObj:=wobjEtna;
